ABB RAPID module: Arm_Weld

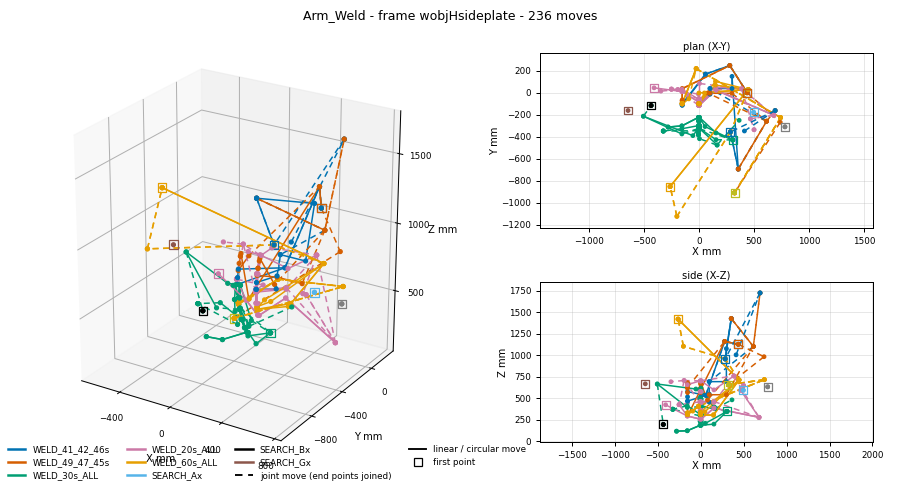
[picture p0: tool path of Arm_Weld in frame wobjHsideplate, 236 of 1587 moves have a stored position in this frame; points joined in program order, loops and branches not executed]
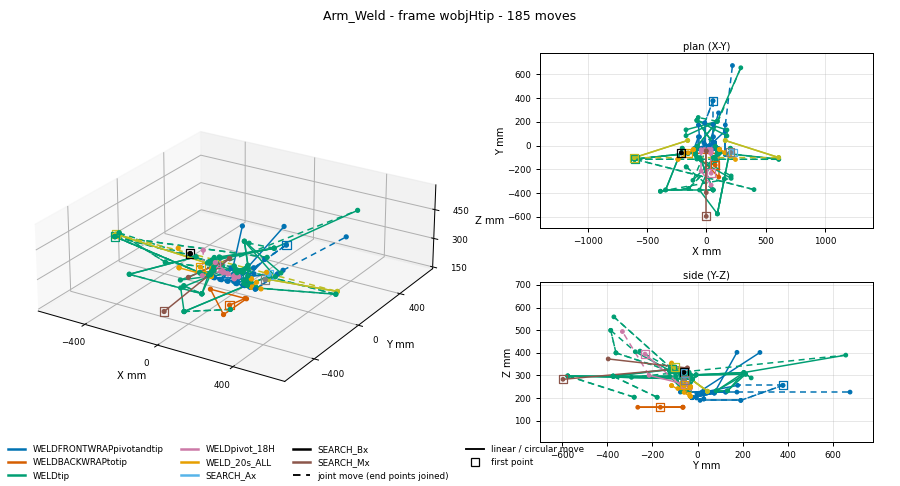
[picture p1: tool path of Arm_Weld in frame wobjHtip, 185 of 1587 moves have a stored position in this frame; points joined in program order, loops and branches not executed]
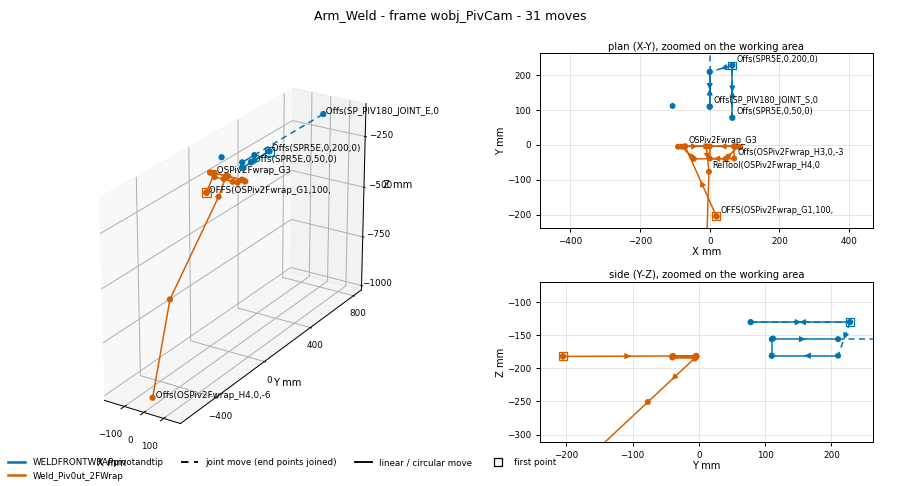
[picture p2: tool path of Arm_Weld in frame wobj_PivCam, 31 of 1587 moves have a stored position in this frame; points joined in program order, loops and branches not executed]
MODULE W6806128_R4_PR3

!!!!!! this is the 7th revision of integrating the NEW PivCAM stuff  SY 12-06-18!!!
!!!!!!THIS IS A PR3 TEMPLATE PROGRAM FOR 18H SIP lesspoints (928)!!!!!03-02-20!!!SY!!!
!!!!!! HAS 3 points 60s!!!
!!!!!!  CAME FROM EMPTY ARM 03-02-20!!!!!!!!
!!!!!! LAYED OUT TO WORK WITH Assembly_Data R12.sys 04-08-18!!!!!!
!!!!!!HAS R100!!04-08-18!!!!!!
!!!!!!!!!BORN FROM 6935130 18H!!!!!!!!
!!!!!!HAS SEARCH_Mx, SEARCH_Lx, SEARCH_Ax, SEARCH_Bx, SEARCH_Gx, SEARCH_Hx!!!!!!!!!!
!!!!!!HAS ZERO_X_A_ALL,ZERO_X_B_ALL,ZERO_X_G_ALL,ZERO_X_H_ALL,ZERO_X_L_ALL,ZERO_X_M_ALL,!!!!!!!!!!
!!!!!!THIS TEMPLATE HAS BEEN REVIEWED IN 5.61  03-02-20!!!!!!!
!!!!!!!!!18H!!!!!!!!!!!!!
!!!!!!!!has FBadjpos/UNtilt19!!! 04-08-18!!!!!
!!!!!!!! HAS TBR/L!04-08-18!!!!!!!!!!!
!!!!!!...04-08-18.now HAS nozzle searching w/IF!!!!!!!
!!!!!!!..anchor is SIP nozzle searching FOR H_ANCHOR,TAPERED_SQUARE_ANCHOR, PLAIN SQUARE ANCHOR....01-09-18!!!!!!!!!!
!!!!!!!Nozzle searching on Anchor is pointing TIP.....(short Wotox)(1012)....08-28-18!!!!!!!!!!
!!!!!!! Fixed a wart in the weld_all_PJ proc....wrong callout in a seamparam in a joint search....03-25-18!!!!
!!!!!!! Created a new x plotter for the anchor (SET_ANCHOR_X) with input 04-08-18
!!!!!!! Created a new x pose SR_AHF_X,SR_AHG_X for the anchor procs  04-08-18
!!!!!!! Created new robtargets  SP_AGFX_E SP_AGFX_S SP_AHFX_E SP_AGFX_S for the anchor procs  04-08-18
!!!!!!! REVISED ALL ANCHOR PROCS TO ADD X SEARCHES ON FRONT and BACK 04-08-18
!!!!!!! ADDED THE PIV PROCs that got Revised 04-08-18
!!!!!!! CUT AND PASTE WELDATA INTO here from template 12-06-18!!!!!!!
!!!!!!! has WELDpivot_18H (only two passes!) 08-16-18!!!!
!!!!!!! now with TWO PASSES ON THE TIP!!!!!!!!!!!!!!!
!!!!!!!HAS dripstop_A and_G with IF...11-27-19!!!!!!!!
!!!!!!! added z_RESETS 04-22-19!!!!!!!!!!!!!!!!!!!!!
!!!!!!!! added ADJWrapperROOTWIDTH18H 11-18-19!!!!!!!!!!!
!!!!!!!!Killed the 0.5 WaitTime in dots in Weldpivot 01-16-20!!!!!!!!
!!!!!!!!!03-02-20 Uses the Revised (R2) Pivot plotter for 18H!!!!!!
!!!!!!!!! 09-28-20 TRACKING HEIGHT ONLY ON ABTBL,ABTBR,GHTBL,GHTBR!!!!!!!!!!




    PERS num scoot_G:=-2.3;
    PERS num scoot_A:=3;

   PERS pose SRRY1:=[[-0.278763,0,0],[1,0,0,0]];

    PERS num THISPROGRAM:=6806128;
    PERS num THISPARTREV:=4;
    PERS num THISPROGREV:=3;
    PERS num THISPROGPREP:=191118;
    VAR bool bSIP:=TRUE;
    VAR bool bINTEGRAL_TIP:=FALSE;
    VAR bool bANC2CLOSE2_TIP:=FALSE;
    VAR bool bBACK_STEP:=FALSE;
    VAR bool bFEEDBACK:=FALSE;
    PERS num THISproglastchanged:=200928;
    VAR bool bUnderANCHOR:=TRUE;
    VAR bool bmissweld:=FALSE;
    VAR num reg100:=0;

!!!!!!!!!!!!!!!!!!!!!!!!!!!!!!!!!  vvvv THESE WELD AND TRACKDATAS COPIED INTO TEMPLATE 11-29-18 vvv !!!!!!!!!!!!!!!!!!!!!!!!!!!!!!!!!!!!
 !!!!!!!!!!!!!!!!WE WILL CALL THIS 18H (8mm) wrapper data!!!!!!!
!!!!!!!!!!dropped current targets to proper values 11-29-18!!!!!!!!!
!!!!!!!!11-29-18!!!!!!!!!!!!


    TASK PERS seamdata smpqroot:=[1,2,[5,5,27.5,135.467,0,325,0,0,0],0,0,0,0,0,[0,0,0,0,0,0,0,0,0],2,0.5,[5,5,27.5,139.7,0,325,0,0,0],0.08,0,[0,0,0,0,0,0,0,0,0],3];
    TASK PERS welddata wdP1Q1root:=[9.31333,0,[5,5,27.5,156.633,0,325,0,0,0],[0,0,0,0,0,0,0,0,0]];

    TASK PERS trackdata trABTBR3:=[0,FALSE,25,[5,40,40,0,-3,0,0,0,0],[0,0,0,0,0,0,0]];
    TASK PERS trackdata trGHTBR3:=[0,FALSE,25,[5,40,40,0,-3,0,0,0,0],[0,0,0,0,0,0,0]];


    PERS num percentcoverpass:=39;
    PERS num percentrootpass:=35;
    PERS num percent2pass:=40;

	TASK PERS trackdata trLM10hiteonly:=[0,FALSE,25,[5,40,40,0,0,0,0,0,0],[0,0,0,0,0,0,0]];

    TASK PERS trackdata trPJhiteonly1:=[0,TRUE,25,[5,40,40,0,0,0,0,0,0],[0,0,0,0,0,0,0]];
    TASK PERS welddata wdGH_CAM_PJ_ROOTfast:=[5.08,0,[5,0,27.8,139.7,0,325,0,0,0],[0,0,0,0,0,0,0,0,0]];
    TASK PERS welddata wdGH_RND_PJ_ROOTfast:=[5.08,0,[5,0,27.8,143.933,0,325,0,0,0],[0,0,0,0,0,0,0,0,0]];
    TASK PERS welddata wdGH_RND_PJ_ROOT:=[3.38667,0,[5,0,27.8,139.7,0,325,0,0,0],[0,0,0,0,0,0,0,0,0]];
    TASK PERS welddata wdGH_CAM_PJ_ROOT:=[3.38667,0,[5,0,27.8,148.167,0,325,0,0,0],[0,0,0,0,0,0,0,0,0]];
    TASK PERS welddata wdGH_RND_PJ_CVR:=[2.96333,0,[5,5,27.5,143.933,0,325,0,0,0],[0,0,0,0,0,0,0,0,0]];

     TASK PERS welddata wdGH_CAM_PJ_FILL1:=[3.38667,0,[5,5,27.8,148.167,0,325,0,0,0],[0,0,0,0,0,0,0,0,0]];
     TASK PERS welddata wdGH_CAM_PJ_FILL2:=[3.38667,0,[5,5,27.8,148.167,0,325,0,0,0],[0,0,0,0,0,0,0,0,0]];
     TASK PERS welddata wdGH_CAM_PJ_CVR:=[3.38667,0,[5,5,27.8,148.167,0,325,0,0,0],[0,0,0,0,0,0,0,0,0]];

     TASK PERS weavedata wvGH_CAM_PJ_FILL2:=[1,0,3,3,0,0.2,0,0.2,0,0,0,0,0,0,0];
     TASK PERS weavedata wvGH_CAM_PJ_FILL1:=[1,0,3,3,0,0.2,0,0.2,0,0,0,0,0,0,0];
     TASK PERS weavedata wvGH_CAM_PJ_CVR:=[1,0,3,3,0,0.2,0,0.2,0,0,0,0,0,0,0];
	 TASK PERS weavedata wvGH_RND_PJ_CVR:=[1,0,5,5,0,0.2,0,0.2,0,0,0,0,0,0,0];

    TASK PERS seamdata smGH_RND_PJ:=[1,2,[5,5,27.8,148.167,0,325,0,0,0],0,1,0,0,0,[0,0,0,0,0,0,0,0,0],1.5,1.3,[5,5,27.8,148.167,0,325,0,0,0],0.08,0,[0,0,0,0,0,0,0,0,0],1];
    TASK PERS seamdata smGH_CAM_PJ:=[1,2,[5,5,27.8,148.167,0,325,0,0,0],0,1,0,0,0,[0,0,0,0,0,0,0,0,0],1.5,1.3,[5,5,27.8,148.167,0,325,0,0,0],0.08,0,[0,0,0,0,0,0,0,0,0],1];

	TASK PERS trackdata trGH:=[0,FALSE,25,[0,40,40,0,0,0,0,0,0],[0,0,0,0,0,0,0]];
	TASK PERS trackdata trAB:=[0,FALSE,25,[0,40,40,0,0,0,0,0,0],[0,0,0,0,0,0,0]];

    TASK PERS trackdata trABTBR:=[0,FALSE,25,[5,40,40,0,-1,0,0,0,0],[0,0,0,0,0,0,0]];
    TASK PERS trackdata trABTBL:=[0,FALSE,25,[5,40,40,0,1,0,0,0,0],[0,0,0,0,0,0,0]];
    TASK PERS trackdata trGHTBR:=[0,FALSE,25,[5,40,40,0,-1,0,0,0,0],[0,0,0,0,0,0,0]];
    TASK PERS trackdata trGHTBL:=[0,FALSE,25,[5,40,40,0,1,0,0,0,0],[0,0,0,0,0,0,0]];


    TASK PERS trackdata trLM18cast:=[0,FALSE,25,[0,40,30,0,0,0,0,0,0],[0,0,0,0,0,0,0]];
    TASK PERS trackdata trTIPears:=[0,FALSE,25,[5,40,40,0,0,0,0,0,0],[0,0,0,0,0,0,0]];
	TASK PERS trackdata trRS56:=[0,TRUE,50,[5,40,40,0,0,0,0,0,0],[0,0,0,0,0,0,0]];
	TASK PERS trackdata trHCYLANCHhiteonly:=[0,TRUE,25,[0,40,40,0,0,0,0,0,0],[0,0,0,0,0,0,0]];
	TASK PERS trackdata track0:=[0,FALSE,0,[0,0,0,0,0,0,0,0,0],[0,0,0,0,0,0,0]];
	TASK PERS trackdata trLM10:=[0,FALSE,25,[0,50,30,0,0,0,0,0,0],[0,0,0,0,0,0,0]];
	TASK PERS trackdata trTIPBACKhiteonly:=[0,TRUE,25,[5,40,40,0,0,0,0,0,0],[0,0,0,0,0,0,0]];

    TASK PERS welddata wdGH195tip:=[6.64633,0,[5,5,26.8,127,0,305,0,0,0],[0,0,0,0,0,0,0,0,0]];
    TASK PERS weavedata wvGH195tip:=[1,0,2,2,0,0,0,0,0,0,0,0,0,0,0];

    TASK PERS welddata wdGH29tip:=[6.68867,0,[5,5,26.8,127,0,305,0,0,0],[0,0,0,0,0,0,0,0,0]];
    TASK PERS weavedata wvGH29tip:=[1,0,2,2,0,0,0,0,0,0,0,0,0,0,0];

	TASK PERS seamdata smGH195:=[1,2,[5,5,27.5,122.767,0,290,0,0,0],0,1,0,0,0,[0,0,0,0,0,0,0,0,0],2,0.8,[5,5,27,122.767,0,290,0,0,0],0.08,0,[0,0,0,0,0,0,0,0,0],2];
	TASK PERS welddata wdGH195:=[6.68867,0,[5,5,26.8,127,0,305,0,0,0],[0,0,0,0,0,0,0,0,0]];
	TASK PERS weavedata wvGH195:=[1,0,2,2,0,0,0,0,0,0,0,0,0,0,0];
	TASK PERS weavedata wvGH29:=[1,0,2,2,0,0,0,0,0,0,0,0,0,0,0];
	TASK PERS seamdata smGH29:=[1,2,[5,5,27.3,122.767,0,290,0,0,0],0,1,0,0,0,[0,0,0,0,0,0,0,0,0],1.3,0.9,[5,5,27,122.767,0,290,0,0,0],0.08,0,[0,0,0,0,0,0,0,0,0],2];
	TASK PERS welddata wdGH29:=[6.68867,0,[5,5,26.8,127,0,305,0,0,0],[0,0,0,0,0,0,0,0,0]];

	TASK PERS welddata wdGH40A:=[5.92667,0,[5,5,27.5,139.7,0,325,0,0,0],[0,0,0,0,0,0,0,0,0]];
	TASK PERS seamdata smGH40A:=[1,2,[5,5,27.5,139.7,0,325,0,0,0],0,1,0,0,0,[0,0,0,0,0,0,0,0,0],3,1,[5,5,27.5,139.7,0,325,0,0,0],0.08,0,[0,0,0,0,0,0,0,0,0],2];
	TASK PERS weavedata wvGH40A:=[1,0,2,2,0,0,0,0,0,0,0,0,0,0,0];

	TASK PERS weavedata wvGH40B:=[1,0,2,2,0,0,0,0,0,0,0,0,0,0,0];
	TASK PERS welddata wdGH40B:=[4.65667,0,[5,5,27.5,139.7,0,325,0,0,0],[0,0,0,0,0,0,0,0,0]];

	TASK PERS welddata wdGH40C:=[7.62,0,[5,5,27.5,143.933,0,325,0,0,0],[0,0,0,0,0,0,0,0,0]];

	TASK PERS welddata wdGH40F:=[7.62,0,[5,0,27.5,131.233,0,300,0,0,0],[0,0,0,0,0,0,0,0,0]];
	TASK PERS seamdata smGH40F:=[1,1,[5,0,27.5,127,0,300,0,0,0],0,1,0,0,0,[0,0,0,0,0,0,0,0,0],1,0,[0,0,0,0,0,0,0,0,0],0,0,[0,0,0,0,0,0,0,0,0],0];

!!!!!!!!!!!!!!!!!BEST 18H weldata and beveldata as of 11-29-18 !!!!!!

	TASK PERS welddata wdR1R2root:=[11.0067,0,[5,5,27.5,152.4,0,320,0,0,0],[0,0,0,0,0,0,0,0,0]];
    TASK PERS weavedata wvRSroot:=[1,0,6,1,0,0,0,0,0,0,0,0,0,0,0];
	TASK PERS welddata wdR5R6cover:=[3.38667,0,[5,5,27.5,143.933,0,325,0,0,0],[0,0,0,0,0,0,0,0,0]];
	TASK PERS welddata wdP1Q1cover:=[4.65667,0,[5,5,27.5,143.933,0,325,0,0,0],[0,0,0,0,0,0,0,0,0]];
	TASK PERS weavedata wvR5R6cover:=[1,0,2,3,0,0.1,0,0.1,0,0,0,0,0,0,0];
	TASK PERS weavedata wvP1Q1cover:=[1,0,2,2,0,0.1,0,0.1,0,20,0,0,0,0,0];
	TASK PERS seamdata smPQRS:=[1,2,[5,5,27.5,148.167,0,320,0,0,0],0,1,0,0,0,[0,0,0,0,0,0,0,0,0],1.2,1.2,[5,5,27.5,139.7,0,320,0,0,0],0.08,0,[0,0,0,0,0,0,0,0,0],1];
	TASK PERS seamdata smPQRSroot:=[1,2,[5,5,27.8,148.167,0,325,0,0,0],0,1,0,0,0,[0,0,0,0,0,0,0,0,0],0,0,[5,5,27.5,127,0,325,0,0,0],0.08,0,[0,0,0,0,0,0,0,0,0],1];
	TASK PERS seamdata smRS1:=[1,2,[5,5,27.5,148.167,0,320,0,0,0],0,1,0,0,0,[0,0,0,0,0,0,0,0,0],1.2,1.2,[5,5,27.5,139.7,0,320,0,0,0],0.08,0,[0,0,0,0,0,0,0,0,0],1];
	TASK PERS seamdata smPQ1:=[1,2,[5,5,27.5,148.167,0,320,0,0,0],0,1,0,0,0,[0,0,0,0,0,0,0,0,0],1.2,1.2,[5,5,27.5,139.7,0,320,0,0,0],0.08,0,[0,0,0,0,0,0,0,0,0],1];

	TASK PERS welddata wdGH1thru8:=[5.50333,0,[5,5,27.5,139.7,0,315,0,0,0],[0,0,0,0,0,0,0,0,0]];
	TASK PERS seamdata smGH1thru8:=[1,2,[5,5,27.5,143.933,0,320,0,0,0],0,1,0,0,0,[0,0,0,0,0,0,0,0,0],1,1.6,[5,5,27.5,143.933,0,320,0,0,0],0.08,0,[0,0,0,0,0,0,0,0,0],1.5];
	TASK PERS weavedata wvGH1thru8:=[1,0,2,2,0,0,0,0,0,0,0,0,0,0,0];

	TASK PERS seamdata smLM10:=[1,2,[5,5,27.5,139.7,0,320,0,0,0],0,1,0,0,0,[0,0,0,0,0,0,0,0,0],1.3,1.2,[5,5,27.5,127,0,320,0,0,0],0.08,0,[0,0,0,0,0,0,0,0,0],1];
	TASK PERS welddata wdLM10:=[5.50333,0,[5,5,27.5,135.467,0,310,0,0,0],[0,0,0,0,0,0,0,0,0]];
	TASK PERS weavedata wvLM10:=[1,0,2,2,0,0,0,0,0,0,0,0,0,0,0];

	TASK PERS seamdata smTU:=[1,2,[5,5,27.5,135.467,0,320,0,0,0],0,1,0,0,0,[0,0,0,0,0,0,0,0,0],1.5,1.5,[5,5,27.5,139.7,0,320,0,0,0],0.08,0,[0,0,0,0,0,0,0,0,0],1.5];
	TASK PERS welddata wdT1112cover:=[4.445,0,[5,5,27.5,143.933,0,325,0,0,0],[0,0,0,0,0,0,0,0,0]];
	TASK PERS weavedata wvT1112cover:=[1,0,2,4,0,0.1,0,0.1,0,0,0,0,0,0,0];

	TASK PERS seamdata smTU2122:=[1,2,[5,5,27.3,148.167,0,325,0,0,0],0,1,0,0,0,[0,0,0,0,0,0,0,0,0],1.5,1,[5,5,27.3,127,0,325,0,0,0],0.08,0,[0,0,0,0,0,0,0,0,0],1];
	TASK PERS welddata wdTU2122cover:=[3.81,0,[5,5,27.75,141.817,0,325,0,0,0],[0,0,0,0,0,0,0,0,0]];
	TASK PERS weavedata wvTU2122cover:=[1,0,2,4,0,0.2,0,0.2,0,0,0,0,0,0,0];


    TASK PERS welddata wdTU3031root:=[6.77333,0,[5,5,27.5,135.467,0,325,0,0,0],[0,0,0,0,0,0,0,0,0]];
	TASK PERS seamdata smTU3031:=[1,2,[5,5,27.5,139.7,0,325,0,0,0],0,1,0,0,0,[0,0,0,0,0,0,0,0,0],3,1.2,[5,5,27.5,139.7,0,325,0,0,0],0.08,0,[0,0,0,0,0,0,0,0,0],2];
	TASK PERS welddata wdTU3031cover:=[2.96333,0,[5,5,27.5,143.933,0,325,0,0,0],[0,0,0,0,0,0,0,0,0]];
	TASK PERS weavedata wvTU3031cover:=[1,0,2,4,0,0.1,0,0.1,0,0,0,0,0,0,0];

    TASK PERS seamdata smTU3031quick:=[1,2,[5,5,27.5,135.467,0,325,0,0,0],0,1,0,0,0,[0,0,0,0,0,0,0,0,0],3,1,[5,5,27.5,135.467,0,325,0,0,0],0.08,0,[0,0,0,0,0,0,0,0,0],1.6];
    TASK PERS welddata wdTU3031quick:=[4.65667,0,[5,5,27.5,143.933,0,325,0,0,0],[0,0,0,0,0,0,0,0,0]];
    TASK PERS weavedata wvTU3031quick:=[1,0,2,2,0,0.2,0,0.2,0,0,0,0,0,0,0];

    TASK PERS seamdata smTU3031quick2:=[1,2,[5,5,27.5,139.7,0,325,0,0,0],0,1,0,0,0,[0,0,0,0,0,0,0,0,0],3,1.2,[5,5,27.5,139.7,0,325,0,0,0],0.08,0,[0,0,0,0,0,0,0,0,0],2];
    TASK PERS welddata wdTU3031quick2:=[3.937,0,[5,5,27.5,143.933,0,325,0,0,0],[0,0,0,0,0,0,0,0,0]];
    TASK PERS weavedata wvTU3031quick2:=[1,0,2,2,0,0,0,0,0,0,0,0,0,0,0];

    TASK PERS welddata wdTU3031quick3:=[3.175,0,[5,5,27.5,143.933,0,325,0,0,0],[0,0,0,0,0,0,0,0,0]];

     TASK PERS welddata wdTU3031SLOW:=[3.38667,0,[5,5,27.5,143.933,0,325,0,0,0],[0,0,0,0,0,0,0,0,0]];
    TASK PERS weavedata wvTU3031SLOW:=[1,0,2,4,0,0,0,0,0,0,0,0,0,0,0];
    TASK PERS seamdata smTU3031SLOW:=[1,2,[5,5,27.5,139.7,0,330,0,0,0],0,1,0,0,0,[0,0,0,0,0,0,0,0,0],3,1.2,[5,5,27.5,139.7,0,325,0,0,0],0.08,0,[0,0,0,0,0,0,0,0,0],2];

	TASK PERS seamdata smT50:=[1,1,[5,0,27,135.467,0,320,0,0,0],0,1,0,0,0,[0,0,0,0,0,0,0,0,0],2,1.2,[5,5,27,139.7,0,325,0,0,0],0,0,[0,0,0,0,0,0,0,0,0],2];
	TASK PERS welddata wdT50:=[4.23333,0,[5,0,27,139.7,0,325,0,0,0],[0,0,0,0,0,0,0,0,0]];
	TASK PERS weavedata wvT50:=[1,0,2,6,0,0,0,0,0,0,0,0,0,0,0];
    TASK PERS welddata wdT50root:=[6.35,0,[5,0,27.5,169.333,0,325,0,0,0],[0,0,0,0,0,0,0,0,0]];

    TASK PERS seamdata smTU7071:=[1,2,[5,5,27.5,148.167,0,320,0,0,0],0,0,0,0,0,[0,0,0,0,0,0,0,0,0],1.5,1.5,[5,5,27.5,143.933,0,325,0,0,0],0.08,0,[0,0,0,0,0,0,0,0,0],1];
    TASK PERS welddata wdTU7071:=[2.96333,0,[5,5,27.5,143.933,0,325,0,0,0],[0,0,0,0,0,0,0,0,0]];
    TASK PERS weavedata wvTU7071:=[1,0,2,3.5,0,0.3,0,0.3,0,0,0,0,0,0,0];

    TASK PERS seamdata smTUroot:=[1,2,[5,5,27,148.167,0,325,0,0,0],0,1,0,0,0,[0,0,0,0,0,0,0,0,0],1.5,0,[5,5,27,139.7,0,325,0,0,0],0.08,0,[0,0,0,0,0,0,0,0,0],1.5];
    TASK PERS welddata wdT1112root:=[8.46667,0,[5,5,27.5,169.333,0,325,0,0,0],[0,0,0,0,0,0,0,0,0]];

	TASK PERS seamdata smHCYLANCH:=[1,2,[5,5,27.5,131.233,0,325,0,0,0],0,1,0,0,0,[0,0,0,0,0,0,0,0,0],1.5,1,[5,5,27.5,127,0,325,0,0,0],0.08,0,[0,0,0,0,0,0,0,0,0],1];
	TASK PERS welddata wdHCYLANCH:=[3.81,0,[5,5,27.5,143.933,0,325,0,0,0],[0,0,0,0,0,0,0,0,0]];
	TASK PERS weavedata wvHCYLANCH:=[1,0,2,2,0,0.1,0,0.1,0,0,0,0,0,0,0];

    PERS edgedata edgedata_HRND_PJ:=[0,8,3,0.052];
    PERS edgedata edgedata_GRND_PJ:=[0,8,3,0.052];
    PERS edgedata edgedata_GCAM_PJ:=[0,8,3,0.052];
    PERS edgedata edgedata_HCAM_PJ:=[0,8,3,0.052];

    TASK PERS seamparam seampar_HRND_PJ:=["H_PJ",0,[42,0.052,339.999,0,0,1,11,0,4,14,-6,2,15,250],202.66,14.4757,14.4757];
    TASK PERS seamparam seampar_GRND_PJ:=["G_PJ",0,[45,0.052,339.999,0,0,1,11,0,4,14,-6,2,15,250],198.028,14.1448,14.1448];
    TASK PERS seamparam seampar_GCAM_PJ:=["G_PJ",0,[40,0.052,148.167,0,0,1,11,0,3,11,-7,2,100,500],179.688,14.7105,10.9592];
    TASK PERS seamparam seampar_HCAM_PJ:=["H_PJ",0,[40,0.052,350.001,0,0,1,11,0,3,11,-7,2,100,500],184.46,15.0514,11.3001];

    PERS bevelparam bevelparam_HRND_pJ:=[6,0,20,0,14,14,0,5,0,0,15,2,2,0.052];
    PERS bevelparam bevelparam_HCAM_pJ:=[4,0,15,0,14,14,0,5,0,0,15,2,2,0.052];
    PERS bevelparam bevelparam_GRND_pj:=[6,0,20,0,14,14,0,5,0,0,15,2,2,0.052];
    PERS bevelparam bevelparam_GCAM_pj:=[4,0,15,0,14,14,0,5,0,0,15,2,2,0.052];

!!!@######################################################################
!  weld datas for the piv "B" weld  18H
    TASK PERS seamdata smJK:=[1,2,[5,5,27.5,139.7,0,325,0,0,0],0,1,0,0,0,[0,0,0,0,0,0,0,0,0],0.5,0.5,[5,5,27.5,127,0,325,0,0,0],0.08,0,[0,0,0,0,0,0,0,0,0],1.2];
    TASK PERS welddata wdJK:=[4.23333,0,[5,5,27.5,143.933,0,325,0,0,0],[0,0,0,0,0,0,0,0,0]];
    TASK PERS weavedata wvJK:=[1,0,2,4,0,0,0,0,0,0,0,0,0,0,0];
    TASK PERS seamdata smJKnofill:=[1,2,[5,5,27.5,139.7,0,325,0,0,0],0,1,0,0,0,[0,0,0,0,0,0,0,0,0],2,0.8,[5,5,27.5,127,0,300,0,0,0],0.08,0,[0,0,0,0,0,0,0,0,0],2];
    TASK PERS welddata wdJK1:=[5.92667,0,[5,5,27.5,135.467,0,330,0,0,0],[0,0,0,0,0,0,0,0,0]];
    TASK PERS seamdata smJK1:=[1,2,[5,5,27.5,139.7,0,330,0,0,0],0,1,0,0,0,[0,0,0,0,0,0,0,0,0],0.5,0.5,[5,5,27.5,127,0,325,0,0,0],0.08,0,[0,0,0,0,0,0,0,0,0],1.2];
    TASK PERS welddata wdJKroot:=[6.77333,0,[5,0,27,131.233,0,310,0,0,0],[0,0,0,0,0,0,0,0,0]];
    TASK PERS seamdata smJKroot:=[2,2,[5,0,27,135.467,0,320,0,0,0],0,1,0,0,0,[0,0,0,0,0,0,0,0,0],2,0,[5,0,0,0,0,0,0,0,0],0,0,[0,0,0,0,0,0,0,0,0],2];
    TASK PERS weavedata wvJKroot:=[1,0,2,1,0,0,0,0,0,0,0,0,0,0,0];


    !!!!!!!!!!!!!!!!!!!!!!!!!!!!!!!!!!Nums for groove searches!!!!!!!!!!!!!!!!!!!!!!!!!!!!!!!!!
VAR num width_T11:=0;
VAR num width_G50:=0;
VAR num width_H50:=0;
VAR num width_RSR1:=0;
VAR num width_PQ1:=0;
VAR num width_T50:=0;
VAR num width_T40:=0;

PERS num Rrootarea:=0;
PERS num GH50rootarea:=0;
VAR num reg7:=0;
VAR num reg8:=0;

PERS edgeresult edgeresultT11:=[[[0.0793076,-0.129463,0.364746],[1,0,0,0]],[[0.0793076,-0.129461,0.364738],[1,0,0,0]],[93.0493,-36.0195,105.505],[93.1546,-28.1059,106.673]];
PERS edgeresult edgeresultT50:=[[[0.0793076,-0.129463,0.364746],[1,0,0,0]],[[0.0793076,-0.129461,0.364738],[1,0,0,0]],[93.0493,-36.0195,105.505],[93.1546,-28.1059,106.673]];
PERS edgeresult edgeresultT40:=[[[0.0793076,-0.129463,0.364746],[1,0,0,0]],[[0.0793076,-0.129461,0.364738],[1,0,0,0]],[93.0493,-36.0195,105.505],[93.1546,-28.1059,106.673]];

PERS bevelparam bevelparamT50:=[8,0,0,0,5,5,0,0,10,0,10,0,0,0.052];
PERS bevelparam bevelparamR1:=[5,0,30,180,8,8,0,0,0,0,5,0,3,0.052];
PERS bevelparam bevelparamA100:=[5,2,2,180,12.7,12.7,0,0,0,0,12.7,0,4,0.052];

PERS edgedata edgedataT55:=[0,8,3,0.052];
PERS edgedata edgedataR10:=[1,8,3,0.052];
PERS edgedata edgedataPQ1:=[0,8,3,0.052];
PERS edgedata edgedataT50:=[0,8,3,0.052];
PERS edgedata edgedataT40:=[0,8,3,0.052];

TASK PERS seamparam seamparT50:=["TWELD",0,[70,0.052,340,0,0,1,11,0,3.5,8,0,2,15,100],82.8542,10.8629,0.862882];
TASK PERS seamparam seamparR1:=["RWELD",0,[80,0.052,340,0,0,1,11,0,2,13,-2,2,25,135],24.4145,5.36121,0.74241];
TASK PERS seamparam seamparS1:=["SWELD",0,[80,0.052,340,0,0,1,11,0,2,13,-2,2,25,135],24.4145,5.36121,0.74241];

TASK PERS layerdata layRWELD:=["RWELD",[78,0.052,340,0,0,1,11,0,0.5,14,0,2,40,125],[1,0,0,0,0,10,0,0,0,0,0,0,[0,0,0,0,0,0]]];
TASK PERS layerdata laySWELD:=["SWELD",[78,0.052,340,0,0,1,11,0,0.5,11,0,2,40,125],[1,0,0,0,0,10,10,0,0,0,0,0,[0,0,0,0,0,0]]];
!!!!!!!!!!!!!!!!!!!!!!!!!!!!!!!!!  ^^^^THESE DATAS COPIED INTO TEMPLATE 11-29-18 PTL ^^^^^^!!!!!!!!!!!!!!!!!!!!!!!!!!!!!!!!!!!!
!!!!!!!!!!!!!!!!!!!!!!!!!!!!!!!!!  ^^^^THESE WELD AND TRACKDATAS COPIED INTO TEMPLATE 11-29-18  ^^^^^^!!!!!!!!!!!!!!!!!!!!!!!!!!!!!!!!!!!!

    !  this rob target is for setting the YZ components of X-Searches
    PERS robtarget PIV_YZ_MASTER_SEARCH:=[[0.08,-16.55,-269.25],[0.410879,-0.609379,0.562263,0.379072],[-1,0,0,0],[9E+09,-0.000202659,0.00203972,9E+09,9E+09,9E+09]];

  !PIVOT_CAM_LOBE
    PERS robtarget H_RND_1:=[[138.75,-56.15,-128.81],[0.791215,-0.426463,-0.392456,0.195157],[-1,1,-2,0],[9E+09,8.53587,-48.4641,9E+09,9E+09,9E+09]];
	PERS robtarget H_RND_2:=[[138.75,-52.19,-134.16],[0.790823,-0.424031,-0.394665,0.197577],[-1,1,-2,0],[9E+09,8.53587,-48.4642,9E+09,9E+09,9E+09]];
	PERS robtarget H_RND_3:=[[138.75,-6.71,-203.72],[0.77354,-0.424849,-0.422397,0.206687],[-1,1,-2,0],[9E+09,8.53592,-48.464,9E+09,9E+09,9E+09]];
	PERS robtarget H_RND_4:=[[138.76,-1.73,-209.20],[0.831387,-0.307692,-0.395259,0.240606],[-1,1,-3,0],[9E+09,8.5359,-60,9E+09,9E+09,9E+09]];
	PERS robtarget H_RND_5:=[[138.77,4.77,-209.99],[0.825767,-0.235199,-0.422961,0.289645],[-1,1,-3,0],[9E+09,17.3096,-65,9E+09,9E+09,9E+09]];
	PERS robtarget H_RND_6:=[[138.76,19.31,-210.84],[0.84569,-0.248028,-0.384006,0.275373],[-1,1,-3,0],[9E+09,17.3096,-67,9E+09,9E+09,9E+09]];
	PERS robtarget H_RND_7:=[[138.75,20.19,-212.40],[0.714518,-0.516691,-0.337745,0.329276],[0,2,-3,0],[9E+09,-11.563,-48.937,9E+09,9E+09,9E+09]];
	PERS robtarget H_RND_8:=[[138.01,1.53,-260.75],[0.775065,-0.4237,-0.381985,0.271739],[-1,2,-3,0],[9E+09,-18.82,-50,9E+09,9E+09,9E+09]];

    PERS robtarget G_RND_1:=[[-137.19,-60.62,-128.24],[0.743875,-0.503842,0.273771,-0.34328],[-1,1,-2,0],[9E+09,8.53587,48.4641,9E+09,9E+09,9E+09]];
	PERS robtarget G_RND_2:=[[-137.17,-55.07,-134.19],[0.733198,-0.515384,0.284408,-0.340458],[-1,1,-2,0],[9E+09,8.53596,48.4639,9E+09,9E+09,9E+09]];
	PERS robtarget G_RND_3:=[[-137.16,-8.79,-203.74],[0.739724,-0.505179,0.29895,-0.328986],[-1,1,-2,0],[9E+09,8.53588,48.4641,9E+09,9E+09,9E+09]];
	PERS robtarget G_RND_4:=[[-137.17,-4.28,-209.04],[0.79307,-0.400763,0.274228,-0.367733],[-1,1,-3,0],[9E+09,8.5359,60,9E+09,9E+09,9E+09]];
	PERS robtarget G_RND_5:=[[-137.17,4.80,-210.46],[0.793114,-0.347997,0.30544,-0.395695],[-1,1,-3,0],[9E+09,17.3096,65,9E+09,9E+09,9E+09]];
	PERS robtarget G_RND_6:=[[-137.17,17.37,-210.42],[0.775238,-0.392589,0.31475,-0.381854],[-1,1,-2,0],[9E+09,17.3096,66.9999,9E+09,9E+09,9E+09]];
	PERS robtarget G_RND_7:=[[-137.15,18.66,-210.61],[0.703635,-0.503523,0.333985,-0.37392],[-1,1,-3,0],[9E+09,-11.563,48.937,9E+09,9E+09,9E+09]];
	PERS robtarget G_RND_8:=[[-137.9,0.7,-261.77],[0.695401,-0.476371,0.308489,-0.440823],[-1,1,-3,0],[9E+09,18.82,50.0001,9E+09,9E+09,9E+09]];

	PERS robtarget G_CAM_1:=[[-92.072,-56.19,-102.39],[0.7891,-0.350678,-0.49169,-0.112189],[-1,1,-2,0],[9E+09,-4.99999,-46.4189,9E+09,9E+09,9E+09]];
	PERS robtarget G_CAM_2:=[[-92.072,-45.7,-130.82],[0.78473,-0.351653,-0.498636,-0.109091],[-1,1,-2,0],[9E+09,-4.99999,-46.4189,9E+09,9E+09,9E+09]];
	PERS robtarget G_CAM_3:=[[-92.072,-38.95,-140.06],[0.856961,-0.220645,-0.451261,-0.115311],[-1,0,-2,0],[9E+09,12,-58,9E+09,9E+09,9E+09]];
	PERS robtarget G_CAM_4:=[[-92.072,-16.92,-148.25],[0.84678,-0.238772,-0.459157,-0.122986],[-1,0,-2,0],[9E+09,14,-60,9E+09,9E+09,9E+09]];
	PERS robtarget G_CAM_5:=[[-92.072,-12.59,-151.76],[0.776964,-0.265744,-0.537769,-0.191078],[-1,0,-2,0],[9E+09,-2.00001,-50.0003,9E+09,9E+09,9E+09]];
	PERS robtarget G_CAM_6:=[[-92.072,-13.07,-165.64],[0.665852,-0.294079,-0.652518,-0.210665],[-1,0,-2,0],[9E+09,-15,-54.9999,9E+09,9E+09,9E+09]];
	PERS robtarget G_CAM_7:=[[-92.072,-12.78,-181.52],[0.705791,-0.252132,-0.619909,-0.232383],[-1,0,-2,0],[9E+09,-18,-54.9998,9E+09,9E+09,9E+09]];
	PERS robtarget G_CAM_8:=[[-92.072,-1.59,-188.14],[0.802926,-0.25985,-0.496077,-0.204193],[-1,0,-2,0],[9E+09,3.00002,-55.0003,9E+09,9E+09,9E+09]];

    PERS robtarget H_CAM_1:=[[98.1522,-58.89,-108.72],[0.766483,-0.505835,0.353281,-0.178403],[-1,1,-2,0],[9E+09,-4.99998,46.581,9E+09,9E+09,9E+09]];
	PERS robtarget H_CAM_2:=[[98.1522,-45.58,-135.58],[0.770116,-0.507654,0.34531,-0.173119],[-1,1,-3,0],[9E+09,-4.99998,46.5812,9E+09,9E+09,9E+09]];
	PERS robtarget H_CAM_3:=[[98.1522,-39.98,-142.01],[0.807219,-0.385353,0.327992,-0.303844],[-1,1,-3,0],[9E+09,12,57.9999,9E+09,9E+09,9E+09]];
	PERS robtarget H_CAM_4:=[[98.1522,-20.35,-148.53],[0.826748,-0.369444,0.308178,-0.291592],[-1,1,-2,0],[9E+09,14,60.0001,9E+09,9E+09,9E+09]];
	PERS robtarget H_CAM_5:=[[98.1522,-10.85,-155.43],[0.769559,-0.521665,0.3083,-0.201484],[-1,1,-2,0],[9E+09,-2.00001,49.9997,9E+09,9E+09,9E+09]];
	PERS robtarget H_CAM_6:=[[98.1522,-14.24,-165.89],[0.659308,-0.625452,0.388751,-0.151641],[-1,1,-2,0],[9E+09,-15,55,9E+09,9E+09,9E+09]];
	PERS robtarget H_CAM_7:=[[98.1522,-15.81,-182.09],[0.670223,-0.62256,0.363504,-0.176309],[-1,1,-2,0],[9E+09,-18,54.9997,9E+09,9E+09,9E+09]];
	PERS robtarget H_CAM_8:=[[98.1522,-3.58,-188.22],[0.796417,-0.486379,0.272771,-0.23399],[-1,1,-3,0],[9E+09,3,54.9999,9E+09,9E+09,9E+09]];

   !!!!!!!!!!!!!
  	PERS robtarget GCam_SidePIV_S:=[[-109.269,-2,-107],[0.649686,-0.594019,0.328892,-0.341878],[-1,1,-2,0],[9E+09,-18.2042,49.7958,9E+09,9E+09,9E+09]];
  	PERS robtarget GCam_SidePIV_Sm:=[[-109.269,-1.99,-117.99],[0.609781,-0.625008,0.349951,-0.339215],[-1,1,-2,0],[9E+09,-18.2042,49.7958,9E+09,9E+09,9E+09]];
  	PERS robtarget GCam_SidePIV_M:=[[-109.269,-2,-140],[0.67995,-0.574742,0.347682,-0.294036],[-1,1,-2,0],[9E+09,-18.2042,49.7958,9E+09,9E+09,9E+09]];
  	PERS robtarget GCam_SidePIV_Em:=[[-109.269,-2,-150],[0.67995,-0.574742,0.347682,-0.294036],[-1,1,-2,0],[9E+09,-18.2042,49.7958,9E+09,9E+09,9E+09]];
  	PERS robtarget GCam_SidePIV_E:=[[-109.269,-0.93,-159.99],[0.618561,-0.622995,0.348237,-0.328618],[-1,1,-2,0],[9E+09,-18.2042,49.7958,9E+09,9E+09,9E+09]];

  	PERS robtarget HCam_SidePIV_S:=[[111.13,1.86,-103.81],[0.654832,-0.57131,-0.34952,0.350194],[-1,2,-3,0],[9E+09,-18.2042,-49.7958,9E+09,9E+09,9E+09]];
  	PERS robtarget HCam_SidePIV_Sm:=[[111.12,1.94,-118.00],[0.631899,-0.613902,-0.344567,0.324192],[-1,2,-3,0],[9E+09,-18.2042,-49.7957,9E+09,9E+09,9E+09]];
  	PERS robtarget HCam_SidePIV_M:=[[111.126,-2,-140],[0.649888,-0.476039,-0.592269,-0.0157843],[-1,1,-2,0],[9E+09,-18.2042,-49.7958,9E+09,9E+09,9E+09]];
  	PERS robtarget HCam_SidePIV_Em:=[[111.126,-2,-150],[0.649888,-0.476039,-0.592269,-0.0157843],[-1,1,-2,0],[9E+09,-18.2042,-49.7958,9E+09,9E+09,9E+09]];
  	PERS robtarget HCam_SidePIV_E:=[[111.13,0.73,-160.00],[0.621633,-0.627968,-0.342345,0.319418],[-1,2,-3,0],[9E+09,-18.2042,-49.7958,9E+09,9E+09,9E+09]];
   !!!!!!!!!!!!!
    PERS pose SRpivotYhelperGsideRound:=[[-0.0176163,-0.000339508,0.049202],[1,0,0,0]];
    PERS robtarget SPpivotYhelperGsideRoundE:=[[-62.04,37.71,-99.13],[0.633362,-0.31447,0.633322,-0.314428],[-1,1,-2,0],[9E+09,5.00002,95,9E+09,9E+09,9E+09]];
    PERS pose SRpivotYhelperHsideRound:=[[0.0116348,-0.255379,-0.025383],[1,0,0,0]];
    PERS robtarget SPpivotYhelperHsideRoundE:=[[62.027,46.7906,-99.2751],[0.690188,-0.153762,-0.69018,0.153784],[-1,1,-2,0],[9E+09,4.99999,-95.0001,9E+09,9E+09,9E+09]];

  	PERS robtarget GRnd_SidePIV_S:=[[-120.769,17.42,-200.71],[0.651172,-0.287913,0.621231,-0.327343],[-1,2,-2,0],[9E+09,5.00002,95,9E+09,9E+09,9E+09]];
  	PERS robtarget GRnd_SidePIV_Sm:=[[-120.769,17.04,-167.64],[0.651174,-0.287913,0.62123,-0.32734],[-1,2,-2,0],[9E+09,5.00002,94.9999,9E+09,9E+09,9E+09]];
  	PERS robtarget GRnd_SidePIV_M:=[[-120.769,17.92,-116.12],[0.651174,-0.287906,0.621235,-0.327337],[-1,2,-2,0],[9E+09,4.99999,95,9E+09,9E+09,9E+09]];
  	PERS robtarget GRnd_SidePIV_Em:=[[-120.769,21.68,-119.15],[0.595995,-0.227597,0.660565,-0.395783],[-1,2,-3,0],[9E+09,4.99999,105,9E+09,9E+09,9E+09]];
  	PERS robtarget GRnd_SidePIV_E:=[[-120.769,17.93,-116.14],[0.65117,-0.287909,0.621236,-0.327341],[-1,2,-2,0],[9E+09,4.99999,95,9E+09,9E+09,9E+09]];

  	PERS robtarget HRnd_SidePIV_S:=[[122.626,21.75,-200.18],[0.703025,-0.151182,-0.677087,0.156371],[-1,1,-2,0],[9E+09,5.00002,-95,9E+09,9E+09,9E+09]];
  	PERS robtarget HRnd_SidePIV_Sm:=[[122.626,21.76,-162.84],[0.703027,-0.151185,-0.677086,0.156368],[-1,1,-2,0],[9E+09,5,-95,9E+09,9E+09,9E+09]];
  	PERS robtarget HRnd_SidePIV_M:=[[122.626,21.76,-119.02],[0.703027,-0.151185,-0.677086,0.156368],[-1,0,-2,0],[9E+09,5,-95,9E+09,9E+09,9E+09]];
  	PERS robtarget HRnd_SidePIV_Em:=[[122.626,28.14,-119.7],[0.681892,-0.000934329,-0.675339,0.280964],[-1,1,-3,0],[9E+09,5,-105,9E+09,9E+09,9E+09]];
  	PERS robtarget HRnd_SidePIV_E:=[[122.626,21.76,-119.02],[0.703027,-0.151185,-0.677086,0.156368],[-1,0,-2,0],[9E+09,5,-95,9E+09,9E+09,9E+09]];
   !!!!!!!!!!!!!!!!!

    PERS robtarget OSPiv2Fwrap_G1:=[[-80.79,-4.98,-182.07],[0.670284,-0.189714,-0.414913,-0.585299],[-1,0,-2,0],[9E+09,21,-0.000317801,9E+09,9E+09,9E+09]];
 	PERS robtarget OSPiv2Fwrap_G2:=[[-91.28,-4.97,-183.63],[0.691634,-0.118244,-0.458469,-0.545405],[-1,0,-3,0],[9E+09,21,-0.000385043,9E+09,9E+09,9E+09]];
  	PERS robtarget OSPiv2Fwrap_G3:=[[-70.80,-3.90,-181.20],[0.644263,-0.288527,-0.274447,-0.652959],[-1,0,-2,0],[9E+09,21,0.00266323,9E+09,9E+09,9E+09]];
  	PERS robtarget OSPiv2Fwrap_G4:=[[0,-3.9,-181.2],[0.644265,-0.28853,-0.274445,-0.652957],[-1,0,-2,0],[9E+09,21,0.00266323,9E+09,9E+09,9E+09]];

 	PERS robtarget OSPiv2Fwrap_H1:=[[80.80,-4.99,-183.81],[0.622109,-0.376532,-0.282896,-0.625439],[-1,0,-2,0],[9E+09,21,0.00302185,9E+09,9E+09,9E+09]];
  	PERS robtarget OSPiv2Fwrap_H2:=[[88.04,-6.32,-185.36],[0.544352,-0.492096,-0.199997,-0.649248],[-1,0,-2,0],[9E+09,21,0.00317875,9E+09,9E+09,9E+09]];
  	PERS robtarget OSPiv2Fwrap_H3:=[[70,-3.88,-182.51],[0.64426,-0.288526,-0.274448,-0.652962],[-1,0,-2,0],[9E+09,21,0.0026184,9E+09,9E+09,9E+09]];
  	PERS robtarget OSPiv2Fwrap_H4:=[[0,-3.88,-182.51],[0.644261,-0.288527,-0.274448,-0.652961],[-1,0,-2,0],[9E+09,21,0.0026184,9E+09,9E+09,9E+09]];

    PERS robtarget SP_Piv0ut_GXs:=[[-31.8,-16.55,-269.25],[0.698471,-0.698472,-0.11017,-0.11017],[-1,0,-2,0],[9E+09,11.5,0,9E+09,9E+09,9E+09]];
 	PERS robtarget SP_Piv0ut_GXe:=[[-81.8,-16.55,-269.25],[0.698471,-0.698472,-0.11017,-0.11017],[-1,0,-2,0],[9E+09,11.5,0,9E+09,9E+09,9E+09]];
    PERS robtarget SP_Piv0ut_HXs:=[[31.8,-16.55,-269.25],[0.705654,-0.705654,-0.0453012,-0.0453012],[-1,1,-2,0],[9E+09,11.5,0,9E+09,9E+09,9E+09]];
    PERS robtarget SP_Piv0ut_HXe:=[[81.8,-16.55,-269.25],[0.705654,-0.705654,-0.0453012,-0.0453012],[-1,1,-2,0],[9E+09,11.5,0,9E+09,9E+09,9E+09]];
    PERS robtarget SP_Piv0ut_Ys:=[[104.208,68.5,960.7],[0.979027,2.38601E-07,5.01456E-08,-0.203733],[-1,2,-4,0],[9E+09,21,0,9E+09,9E+09,9E+09]];
    PERS robtarget SP_Piv0ut_Ye:=[[104.208,13.5,960.7],[0.979027,2.38601E-07,5.01456E-08,-0.203733],[-1,2,-4,0],[9E+09,21,0,9E+09,9E+09,9E+09]];
    PERS robtarget SP_Piv0ut_Zs:=[[104.208,36,994.2],[0.680616,-0.680616,0.191734,0.191734],[-1,1,-2,0],[9E+09,21,0,9E+09,9E+09,9E+09]];
    PERS robtarget SP_Piv0ut_Ze:=[[104.208,36,944.2],[0.680616,-0.680616,0.191734,0.191734],[-1,1,-2,0],[9E+09,21,0,9E+09,9E+09,9E+09]];

!!!!!!!!!!!!!!!!!!!!!!!!!!!!!!!!!!!!!!!!!!!!!!added 03-19-18!!!!!!!!!!!!!!!!!!!!!!!!!!!!!!!!!!!!!!!!
    PERS robtarget SP_YPIVadj_e:=[[0.86,2.59,-78.86],[0.69905,-0.106585,-0.106578,-0.699006],[-1,0,-2,0],[9E+09,21,8.56463E-05,9E+09,9E+09,9E+09]];
    PERS robtarget SP_ZPIVadj_e:=[[-17.01,-7.87,-179.30],[0.669714,-0.669689,-0.226944,-0.226928],[-1,1,-2,0],[9E+09,21,0.00064599,9E+09,9E+09,9E+09]];
    PERS pose SR_YPIVadj:=[[-0.033515,-0.692593,0.000984192],[1,0,0,0]];
    PERS pose SR_ZPIVadj:=[[-0.00343895,-0.541453,-1.49567],[1,0,0,0]];
!!!!!!!!!!!!!!!!!!!!!!!!!!!!!!!!!!!!!!!!!!!!!!!!!!!!!!!!!!!!!!!!!!!!!!!!!!!!!!!!!!!!!!!!!!!!!!!!!!!!!
!!!!!!!!!!!!!!!!!!!!!!!!!!!!!!!!!!!!!!!!!!!!!!!!!!!!!!!!!!!!!!!!!!!!!!!!!!!!!!!!!!!!!!!!!!!!!!!!!!!!!!!!!!!!!!!!!!!
!!        PJ = Pivot Joint   these are for the round shaped pivots
 	PERS robtarget G_PJRnd_1st_s:=[[-116.221,-56.77,-124],[0.71687,-0.11073,-0.684807,-0.0698286],[-1,-2,0,1],[9E+09,5,-90,9E+09,9E+09,9E+09]];
 	PERS robtarget G_PJRnd_1st_sm:=[[-116.221,-46.92,-125.74],[0.71687,-0.11073,-0.684807,-0.0698286],[-1,-2,0,1],[9E+09,5,-90,9E+09,9E+09,9E+09]];
 	PERS robtarget G_PJRnd_1st_em:=[[-116.221,6.76,-136.16],[0.731336,-0.185377,-0.643337,-0.129998],[-1,-2,0,1],[9E+09,5,-90,9E+09,9E+09,9E+09]];
 	PERS robtarget G_PJRnd_1st_e:=[[-116.221,16.76,-137],[0.744449,-0.19541,-0.62012,-0.151862],[-1,-2,0,1],[9E+09,5,-90,9E+09,9E+09,9E+09]];

 	PERS robtarget G_PJRnd_2nd_s:=[[-116.221,-56.77,-124],[0.71687,-0.110731,-0.684806,-0.0698332],[-1,-2,0,1],[9E+09,4.99997,-84.9999,9E+09,9E+09,9E+09]];
 	PERS robtarget G_PJRnd_2nd_sm:=[[-116.221,-46.92,-125.74],[0.71687,-0.11073,-0.684807,-0.0698286],[-1,-2,0,1],[9E+09,5,-85,9E+09,9E+09,9E+09]];
 	PERS robtarget G_PJRnd_2nd_em:=[[-116.221,6.76,-136.16],[0.756184,-0.180674,-0.614904,-0.132046],[-1,-2,0,1],[9E+09,4.99768,-85,9E+09,9E+09,9E+09]];
 	PERS robtarget G_PJRnd_2nd_e:=[[-116.221,16.76,-137],[0.761618,-0.196052,-0.599226,-0.149766],[-1,-2,0,1],[9E+09,4.99767,-74.9999,9E+09,9E+09,9E+09]];

 	PERS robtarget G_PJRnd_3rd_s:=[[-116.221,-56.77,-124],[0.71687,-0.11073,-0.684807,-0.0698286],[-1,-2,0,1],[9E+09,5,-85,9E+09,9E+09,9E+09]];
 	PERS robtarget G_PJRnd_3rd_sm:=[[-116.221,-46.92,-125.74],[0.71687,-0.11073,-0.684807,-0.0698286],[-1,-2,0,1],[9E+09,5,-85,9E+09,9E+09,9E+09]];
 	PERS robtarget G_PJRnd_3rd_em:=[[-116.221,6.76,-136.16],[0.759108,-0.156585,-0.621504,-0.11388],[-1,-2,0,1],[9E+09,5,-85,9E+09,9E+09,9E+09]];
 	PERS robtarget G_PJRnd_3rd_e:=[[-116.221,16.76,-137],[0.690713,-0.364323,-0.609662,-0.136004],[-1,-2,1,1],[9E+09,5,-85,9E+09,9E+09,9E+09]];

 	PERS robtarget G_PJRnd_4th_s:=[[-116.221,-56.77,-124],[0.71687,-0.11073,-0.684807,-0.0698286],[-1,-2,0,1],[9E+09,5,-85,9E+09,9E+09,9E+09]];
 	PERS robtarget G_PJRnd_4th_sm:=[[-116.221,-46.92,-125.74],[0.71687,-0.11073,-0.684807,-0.0698286],[-1,-2,0,1],[9E+09,5,-85,9E+09,9E+09,9E+09]];
 	PERS robtarget G_PJRnd_4th_em:=[[-116.221,6.76,-136.16],[0.759108,-0.156585,-0.621504,-0.11388],[-1,-2,0,1],[9E+09,5,-85,9E+09,9E+09,9E+09]];
 	PERS robtarget G_PJRnd_4th_e:=[[-116.221,16.76,-137],[0.690713,-0.364323,-0.609662,-0.136004],[-1,-2,1,1],[9E+09,5,-85,9E+09,9E+09,9E+09]];

 	PERS robtarget H_PJRnd_1st_s:=[[116.85,-50.63,-124.76],[0.645351,-0.379915,0.599982,-0.28144],[-1,1,2,0],[9E+09,4.99999,90.0002,9E+09,9E+09,9E+09]];
 	PERS robtarget H_PJRnd_1st_sm:=[[116.84,-40.53,-125.74],[0.633823,-0.410174,0.57585,-0.313723],[-1,1,2,0],[9E+09,4.99999,90.0001,9E+09,9E+09,9E+09]];
 	PERS robtarget H_PJRnd_1st_em:=[[116.84,-1.05,-133.41],[0.656479,-0.48509,0.443945,-0.369643],[-1,1,2,0],[9E+09,4.99999,90,9E+09,9E+09,9E+09]];
 	PERS robtarget H_PJRnd_1st_e:=[[116.85,12.27,-135.78],[0.684689,-0.478579,0.414268,-0.361309],[-1,1,1,0],[9E+09,4.99999,90,9E+09,9E+09,9E+09]];

 	PERS robtarget H_PJRnd_2nd_s:=[[116.84,-52.58,-123.26],[0.668155,-0.357654,0.579241,-0.300222],[-1,1,2,0],[9E+09,4.99999,84.9999,9E+09,9E+09,9E+09]];
 	PERS robtarget H_PJRnd_2nd_sm:=[[116.86,-41.60,-125.09],[0.668503,-0.394742,0.522148,-0.35305],[-1,1,2,0],[9E+09,5.00003,85,9E+09,9E+09,9E+09]];
 	PERS robtarget H_PJRnd_2nd_em:=[[116.848,0.57,-132.97],[0.690657,-0.443246,0.412829,-0.395092],[-1,1,1,0],[9E+09,4.99997,84.9999,9E+09,9E+09,9E+09]];
 	PERS robtarget H_PJRnd_2nd_e:=[[117.21,10.44,-135.86],[0.701835,-0.479653,0.380667,-0.36394],[-1,1,1,0],[9E+09,4.99997,75,9E+09,9E+09,9E+09]];

 	PERS robtarget H_PJRnd_3rd_s:=[[116.848,-56.77,-124],[0.645356,-0.379913,0.59998,-0.281436],[-1,1,2,0],[9E+09,5,85,9E+09,9E+09,9E+09]];
 	PERS robtarget H_PJRnd_3rd_sm:=[[116.848,-46.92,-125.74],[0.625682,-0.424599,0.565304,-0.32965],[-1,1,2,0],[9E+09,5,85,9E+09,9E+09,9E+09]];
 	PERS robtarget H_PJRnd_3rd_em:=[[116.848,6.76,-136.16],[0.653344,-0.494982,0.443626,-0.362395],[-1,1,2,0],[9E+09,5,85,9E+09,9E+09,9E+09]];
 	PERS robtarget H_PJRnd_3rd_e:=[[116.848,16.76,-137],[0.681465,-0.518041,0.399083,-0.32859],[-1,1,2,0],[9E+09,5,85,9E+09,9E+09,9E+09]];

 	PERS robtarget H_PJRnd_4th_s:=[[112.848,-56.77,-124],[0.645356,-0.379913,0.59998,-0.281436],[-1,1,2,0],[9E+09,5,85,9E+09,9E+09,9E+09]];
 	PERS robtarget H_PJRnd_4th_sm:=[[112.848,-46.92,-125.74],[0.625682,-0.424599,0.565304,-0.32965],[-1,1,2,0],[9E+09,5,85,9E+09,9E+09,9E+09]];
 	PERS robtarget H_PJRnd_4th_em:=[[112.848,6.76,-136.16],[0.653344,-0.494982,0.443626,-0.362395],[-1,1,2,0],[9E+09,5,85,9E+09,9E+09,9E+09]];
 	PERS robtarget H_PJRnd_4th_e:=[[110.848,16.76,-137],[0.681465,-0.518041,0.399083,-0.32859],[-1,1,2,0],[9E+09,5,85,9E+09,9E+09,9E+09]];

!!!!!!!!!!!!!!!!!!!!!!!!!!!!!!!!!!!!!!!!!!!!!!!!!!!!!!!!!!!!!!!!!!!!!!!!!!!!!!!!!!!!!!!!!!!!!!!!!!!!!!!!!!!!!!!!!!!!!!!!!!!!!!!!!
!!        PJ = Pivot Joint   these are for the CAM shaped pivots
 	PERS robtarget H_PJCam_1st_s:=[[110.602,-2.4,-110.82],[0.398951,-0.65704,-0.250921,0.588367],[-1,-3,3,1],[9E+09,4.67604E-05,-90.0002,9E+09,9E+09,9E+09]];
	PERS robtarget H_PJCam_1st_sm:=[[110.602,-5.8,-110.15],[0.318277,-0.633541,-0.321425,0.627703],[-1,-4,3,1],[9E+09,-4.98748E-06,-90,9E+09,9E+09,9E+09]];
	PERS robtarget H_PJCam_1st_em:=[[110.602,-44.04,-99.16],[0.309721,-0.615411,-0.329677,0.645488],[-1,-4,3,1],[9E+09,5.73674E-05,-90.0003,9E+09,9E+09,9E+09]];
	PERS robtarget H_PJCam_1st_e:=[[110.602,-51.33,-96.68],[0.301369,-0.599085,-0.337318,0.660675],[-1,-4,3,1],[9E+09,3.65824E-05,-90.0001,9E+09,9E+09,9E+09]];

	PERS robtarget H_PJCam_2nd_s:=[[110.602,-1,-111.55],[0.398955,-0.657033,-0.250926,0.58837],[-1,-3,3,1],[9E+09,5,-90,9E+09,9E+09,9E+09]];
	PERS robtarget H_PJCam_2nd_sm:=[[110.602,-5.79,-110.26],[0.318281,-0.633538,-0.321426,0.627704],[-1,-4,3,1],[9E+09,5,-90,9E+09,9E+09,9E+09]];
	PERS robtarget H_PJCam_2nd_em:=[[110.602,-45.58,-99.59],[0.309717,-0.615414,-0.32968,0.645486],[-1,-4,3,1],[9E+09,5,-90,9E+09,9E+09,9E+09]];
    PERS robtarget H_PJCam_2nd_e:=[[110.602,-50.41,-98.3],[0.306036,-0.582148,-0.33034,0.676994],[-1,-4,3,1],[9E+09,5,-90,9E+09,9E+09,9E+09]];

 	PERS robtarget H_PJCam_3rd_s:=[[110.602,-1,-111.55],[0.398955,-0.657033,-0.250926,0.58837],[-1,-3,3,1],[9E+09,5,-90,9E+09,9E+09,9E+09]];
	PERS robtarget H_PJCam_3rd_sm:=[[110.602,-5.79,-110.26],[0.318281,-0.633538,-0.321426,0.627704],[-1,-4,3,1],[9E+09,5,-90,9E+09,9E+09,9E+09]];
	PERS robtarget H_PJCam_3rd_em:=[[110.602,-45.58,-99.59],[0.309717,-0.615414,-0.32968,0.645486],[-1,-4,3,1],[9E+09,5,-90,9E+09,9E+09,9E+09]];
    PERS robtarget H_PJCam_3rd_e:=[[110.602,-50.41,-98.3],[0.306036,-0.582148,-0.33034,0.676994],[-1,-4,3,1],[9E+09,5,-90,9E+09,9E+09,9E+09]];

	PERS robtarget H_PJCam_4th_s:=[[110.602,-1.71,-111.68],[0.42228,-0.640978,-0.232213,0.597415],[-1,-3,3,1],[9E+09,2.59754E-05,-90,9E+09,9E+09,9E+09]];
	PERS robtarget H_PJCam_4th_sm:=[[110.602,-7.26,-110.35],[0.358651,-0.636258,-0.280366,0.622848],[-1,-4,3,1],[9E+09,-5.20202E-06,-90,9E+09,9E+09,9E+09]];
	PERS robtarget H_PJCam_4th_em:=[[110.602,-46.66,-100.15],[0.343263,-0.630093,-0.29504,0.630955],[-1,-4,3,1],[9E+09,2.59754E-05,-89.9999,9E+09,9E+09,9E+09]];
    PERS robtarget H_PJCam_4th_e:=[[110.602,-55.59,-97.87],[0.348944,-0.623408,-0.28586,0.638659],[-1,-4,3,1],[9E+09,-4.67719E-05,-90,9E+09,9E+09,9E+09]];

	PERS robtarget H_PJCam_5th_s:=[[110.602,-6.5,-156.6],[0.39895,-0.657033,-0.250928,0.588372],[-1,-3,3,1],[9E+09,5,-90,9E+09,9E+09,9E+09]];
	PERS robtarget H_PJCam_5th_sm:=[[110.602,-11.35,-154.75],[0.318286,-0.633538,-0.321426,0.627702],[-1,-4,3,1],[9E+09,5,-90,9E+09,9E+09,9E+09]];
	PERS robtarget H_PJCam_5th_em:=[[110.602,-67.65,-139.8],[0.309714,-0.615412,-0.329681,0.645489],[-1,-4,3,1],[9E+09,5,-90,9E+09,9E+09,9E+09]];
	PERS robtarget H_PJCam_5th_e:=[[110.602,-72.5,-138.5],[0.306033,-0.58215,-0.330337,0.676995],[-1,-4,3,1],[9E+09,5,-90,9E+09,9E+09,9E+09]];

 	PERS robtarget G_PJCam_1st_s:=[[-107.775,-5.82,-110.51],[0.664139,-0.454628,0.507295,-0.308033],[-1,1,-2,0],[9E+09,-0.000171267,90.0005,9E+09,9E+09,9E+09]];
	PERS robtarget G_PJCam_1st_sm:=[[-107.775,-9.93,-108.79],[0.599292,-0.389593,0.57554,-0.397266],[-1,1,-2,0],[9E+09,-4.98748E-06,89.9999,9E+09,9E+09,9E+09]];
	PERS robtarget G_PJCam_1st_em:=[[-107.775,-47.4,-97.95],[0.58619,-0.377085,0.588845,-0.409206],[-1,1,-2,0],[9E+09,2.59754E-05,90.0001,9E+09,9E+09,9E+09]];
    PERS robtarget G_PJCam_1st_e:=[[-107.775,-52.34,-97.4],[0.585528,-0.365611,0.587357,-0.422489],[-1,1,-2,0],[9E+09,-4.67719E-05,89.9999,9E+09,9E+09,9E+09]];

	PERS robtarget G_PJCam_2nd_s:=[[-107.775,-1,-111.55],[0.664146,-0.454653,0.507271,-0.30802],[-1,1,-2,0],[9E+09,5,90,9E+09,9E+09,9E+09]];
	PERS robtarget G_PJCam_2nd_sm:=[[-107.775,-5.79,-110.26],[0.606546,-0.394607,0.567886,-0.392291],[-1,1,-2,0],[9E+09,5,90,9E+09,9E+09,9E+09]];
	PERS robtarget G_PJCam_2nd_em:=[[-107.775,-45.58,-99.59],[0.599356,-0.386244,0.575437,-0.400574],[-1,1,-2,0],[9E+09,5,90,9E+09,9E+09,9E+09]];
	PERS robtarget G_PJCam_2nd_e:=[[-107.775,-50.41,-98.3],[0.585534,-0.365613,0.58735,-0.422489],[-1,1,-2,0],[9E+09,5,90,9E+09,9E+09,9E+09]];

 	PERS robtarget G_PJCam_3rd_s:=[[-107.775,-1,-111.55],[0.664146,-0.454653,0.507271,-0.30802],[-1,1,-2,0],[9E+09,5,90,9E+09,9E+09,9E+09]];
	PERS robtarget G_PJCam_3rd_sm:=[[-107.775,-5.79,-110.26],[0.606546,-0.394607,0.567886,-0.392291],[-1,1,-2,0],[9E+09,5,90,9E+09,9E+09,9E+09]];
	PERS robtarget G_PJCam_3rd_em:=[[-107.775,-45.58,-99.59],[0.599356,-0.386244,0.575437,-0.400574],[-1,1,-2,0],[9E+09,5,90,9E+09,9E+09,9E+09]];
    PERS robtarget G_PJCam_3rd_e:=[[-107.775,-50.41,-98.3],[0.585534,-0.365613,0.58735,-0.422489],[-1,1,-2,0],[9E+09,5,90,9E+09,9E+09,9E+09]];

	PERS robtarget G_PJCam_4th_s:=[[-107.775,-4.09,-111.57],[0.668527,-0.451948,0.50314,-0.309297],[-1,1,-2,0],[9E+09,-0.000399902,89.9987,9E+09,9E+09,9E+09]];
	PERS robtarget G_PJCam_4th_sm:=[[-107.775,-9.52,-111.1],[0.610875,-0.406949,0.562731,-0.380207],[-1,1,-2,0],[9E+09,-5.69499E-05,89.9997,9E+09,9E+09,9E+09]];
	PERS robtarget G_PJCam_4th_em:=[[-107.775,-47.67,-100.86],[0.60677,-0.402434,0.567094,-0.385073],[-1,1,-2,0],[9E+09,-5.69499E-05,89.9998,9E+09,9E+09,9E+09]];
	PERS robtarget G_PJCam_4th_e:=[[-107.775,-57.31,-99.48],[0.597922,-0.371998,0.574618,-0.417038],[-1,1,-3,0],[9E+09,-4.98748E-06,89.9999,9E+09,9E+09,9E+09]];

	PERS robtarget G_PJCam_5th_s:=[[-107.775,-6.5,-156.6],[0.664146,-0.454652,0.507271,-0.308022],[-1,1,-2,0],[9E+09,5,90,9E+09,9E+09,9E+09]];
	PERS robtarget G_PJCam_5th_sm:=[[-107.775,-11.35,-154.75],[0.606547,-0.39461,0.567882,-0.392293],[-1,1,-2,0],[9E+09,5,90,9E+09,9E+09,9E+09]];
	PERS robtarget G_PJCam_5th_em:=[[-107.775,-67.65,-139.8],[0.599352,-0.386244,0.575442,-0.400573],[-1,1,-2,0],[9E+09,5,90,9E+09,9E+09,9E+09]];
	PERS robtarget G_PJCam_5th_e:=[[-107.775,-72.5,-138.5],[0.615886,-0.387535,0.555435,-0.402483],[-1,1,-2,0],[9E+09,5,90,9E+09,9E+09,9E+09]];


    !!!!!!!!!!!!!!!!!!!!!!!!!!!!!!!!!!!!!!!!!!!!!!!!!!!!!!!!!!!!!!!!!!!!!!!!!!!!!!!!!!!!!!!!!!!!!!!!!!!!!!!!!!!!!!!!!!!!!!!!!!!!!
    !!!    SEARCHES FOR G/H PIV 1 THRU 8
    !!!!!!!!!!!!!!!!!!!!!!!!!!!!!!!!!!!!!!!!!!!!!!!!!!!!!!!!!!!!!!!!!!!!!!!!!!!!!!!!!!!!!!!!!!!!!!!!!!!!!!!!!!!!!!!!!!!!!!!!!!
  !!        18 = points 1 thru 8, in CAM or RND Pivots
    PERS robtarget SP_gPivRnd_18_Xs:=[[-158.8,-16.55,-269.25],[0.074768,-0.0747681,-0.703143,-0.703143],[-1,0,-3,0],[9E+09,8.5359,48.4641,9E+09,9E+09,9E+09]];
 	PERS robtarget SP_gPivRnd_18_Xe:=[[-108.8,-16.55,-269.25],[0.074768,-0.0747681,-0.703143,-0.703143],[-1,0,-3,0],[9E+09,8.5359,48.4641,9E+09,9E+09,9E+09]];
 	PERS robtarget SP_hPivRnd_18_Xs:=[[158.8,-16.55,-269.25],[0.6019,-0.601901,-0.371101,-0.3711],[-1,0,-1,0],[9E+09,8.5359,-48.4641,9E+09,9E+09,9E+09]];
 	PERS robtarget SP_hPivRnd_18_Xe:=[[108.8,-16.55,-269.25],[0.6019,-0.601901,-0.371101,-0.3711],[-1,0,-1,0],[9E+09,8.5359,-48.4641,9E+09,9E+09,9E+09]];

    PERS robtarget SP_gPivCam_18_Xs:=[[-31.8,-16.55,-269.25],[0.669176,-0.669177,-0.228479,-0.228479],[-1,0,-1,0],[9E+09,0,-45,9E+09,9E+09,9E+09]];
 	PERS robtarget SP_gPivCam_18_Xe:=[[-81.8,-16.55,-269.25],[0.669176,-0.669177,-0.228479,-0.228479],[-1,0,-1,0],[9E+09,0,-45,9E+09,9E+09,9E+09]];
 	PERS robtarget SP_hPivCam_18_Xs:=[[31.8,-16.55,-269.25],[0.228057,-0.228057,-0.669321,-0.66932],[-1,0,-3,0],[9E+09,0,45,9E+09,9E+09,9E+09]];
 	PERS robtarget SP_hPivCam_18_Xe:=[[81.8,-16.55,-269.25],[0.228057,-0.228057,-0.669321,-0.66932],[-1,0,-3,0],[9E+09,0,45,9E+09,9E+09,9E+09]];

 	PERS robtarget SP_HPivRND_18_Ys:=[[134.755,63.5,811.2],[7.62829E-08,-0.962536,0.271153,1.37778E-07],[-1,1,-2,0],[9E+09,8.5359,-48.4641,9E+09,9E+09,9E+09]];
 	PERS robtarget SP_HPivRND_18_Ye:=[[134.755,13.5,811.2],[7.62829E-08,-0.962536,0.271153,1.37778E-07],[-1,1,-2,0],[9E+09,8.5359,-48.4641,9E+09,9E+09,9E+09]];
 	PERS robtarget SP_HPivRND_18_Zs:=[[134.755,25,977.2],[0.680616,-0.680616,0.191734,0.191734],[-1,-1,0,0],[9E+09,8.5359,-48.4641,9E+09,9E+09,9E+09]];
 	PERS robtarget SP_HPivRND_18_Ze:=[[134.755,25,942.2],[0.680616,-0.680616,0.191734,0.191734],[-1,-1,0,0],[9E+09,8.5359,-48.4641,9E+09,9E+09,9E+09]];

 	PERS robtarget SP_GPivRND_18_Ys:=[[-133.168,63.5,833.7],[3.37488E-07,0.324654,-0.945833,3.78335E-08],[-1,0,0,0],[9E+09,8.5359,48.4641,9E+09,9E+09,9E+09]];
 	PERS robtarget SP_GPivRND_18_Ye:=[[-133.168,13.5,833.7],[3.37488E-07,0.324654,-0.945833,3.78335E-08],[-1,0,0,0],[9E+09,8.5359,48.4641,9E+09,9E+09,9E+09]];
 	PERS robtarget SP_GPivRND_18_Zs:=[[-133.168,25,977.2],[0.229565,-0.229565,0.668805,0.668805],[0,-1,2,0],[9E+09,8.5359,48.4641,9E+09,9E+09,9E+09]];
 	PERS robtarget SP_GPivRND_18_Ze:=[[-133.168,25,942.2],[0.229565,-0.229565,0.668805,0.668805],[0,-1,2,0],[9E+09,8.5359,48.4641,9E+09,9E+09,9E+09]];

  	PERS robtarget SP_HPivCAM_18_Ys:=[[108.152,63.5,826.2],[7.62829E-08,-0.962536,0.271153,1.37778E-07],[-1,1,-2,0],[9E+09,0,45,9E+09,9E+09,9E+09]];
 	PERS robtarget SP_HPivCAM_18_Ye:=[[108.152,13.5,826.2],[7.62829E-08,-0.962536,0.271153,1.37778E-07],[-1,1,-2,0],[9E+09,0,45,9E+09,9E+09,9E+09]];
 	PERS robtarget SP_HPivCAM_18_Zs:=[[108.152,25,977.2],[0.646945,-0.646944,0.285416,0.285418],[-1,2,-2,0],[9E+09,0,45,9E+09,9E+09,9E+09]];
 	PERS robtarget SP_HPivCAM_18_Ze:=[[108.152,25,942.2],[0.646944,-0.646947,0.285414,0.285417],[-1,2,-2,0],[9E+09,0,45,9E+09,9E+09,9E+09]];

 	PERS robtarget SP_GPivCAM_18_Ys:=[[-98.072,63.5,953.7],[0.918423,-1.83184E-08,6.48462E-09,0.3956],[-1,0,-1,1],[9E+09,0,-45,9E+09,9E+09,9E+09]];
 	PERS robtarget SP_GPivCAM_18_Ye:=[[-98.072,13.5,953.7],[0.918423,-1.83184E-08,6.48462E-09,0.3956],[-1,0,-1,1],[9E+09,0,-45,9E+09,9E+09,9E+09]];
 	PERS robtarget SP_GPivCAM_18_Zs:=[[-98.072,25,977.2],[0.703252,-0.703252,-0.0737343,-0.0737346],[-1,0,-1,0],[9E+09,0,-45,9E+09,9E+09,9E+09]];
 	PERS robtarget SP_GPivCAM_18_Ze:=[[-98.072,25,942.2],[0.703252,-0.703252,-0.0737343,-0.0737346],[-1,0,-1,0],[9E+09,0,-45,9E+09,9E+09,9E+09]];

    !!!!!!!!!!!!!!!!!!!!!!!!!!!!!!!!!!!!!!!!!!!!!!!!!!!!!!!!!!!!!!!!!!!!!!!!!!!!!!!!!!!!!!!!!!!!!!!!!!!!!!!!!!!!!!!!!!!!!!!!!!!!!
    !!!    SEARCHES FOR G/H           PJ = PIVOT JOINT            !!!
    !!!!!!!!!!!!!!!!!!!!!!!!!!!!!!!!!!!!!!!!!!!!!!!!!!!!!!!!!!!!!!!!!!!!!!!!!!!!!!!!!!!!!!!!!!!!!!!!!!!!!!!!!!!!!!!!!!!!!!!!!!

    PERS robtarget SP_gPivRnd_PJ_Xs:=[[-19.8,-16.55,-269.25],[0.671032,-0.741422,0.00221101,0.00200072],[-1,0,-1,0],[9E+09,5,-60,9E+09,9E+09,9E+09]];
 	PERS robtarget SP_gPivRnd_PJ_Xe:=[[-69.8,-16.55,-269.25],[0.671032,-0.741422,0.00221101,0.00200072],[-1,0,-1,0],[9E+09,5,-60,9E+09,9E+09,9E+09]];
 	PERS robtarget SP_hPivRnd_PJ_Xs:=[[19.8,-16.55,-269.25],[0.0441236,-0.0785833,-0.868404,-0.487598],[-1,1,0,0],[9E+09,5,90,9E+09,9E+09,9E+09]];
 	PERS robtarget SP_hPivRnd_PJ_Xe:=[[69.8,-16.55,-269.25],[0.0441236,-0.0785833,-0.868404,-0.487598],[-1,1,0,0],[9E+09,5,90,9E+09,9E+09,9E+09]];

    PERS robtarget SP_gPivCam_PJ_Xs:=[[-170.8,-16.55,-269.25],[0.0596632,-0.110181,-0.872423,-0.472418],[-1,-2,-2,1],[9E+09,0,90,9E+09,9E+09,9E+09]];
 	PERS robtarget SP_gPivCam_PJ_Xe:=[[-120.8,-16.55,-269.25],[0.0596632,-0.110181,-0.872423,-0.472418],[-1,-2,-2,1],[9E+09,0,90,9E+09,9E+09,9E+09]];
 	PERS robtarget SP_hPivCam_PJ_Xs:=[[170.8,-16.55,-269.25],[0.981346,-0.071223,0.0129263,0.1781],[0,-1,-1,0],[9E+09,0,-90,9E+09,9E+09,9E+09]];
 	PERS robtarget SP_hPivCam_PJ_Xe:=[[120.8,-16.55,-269.25],[0.981346,-0.071223,0.0129263,0.1781],[0,-1,-1,0],[9E+09,0,-90,9E+09,9E+09,9E+09]];

 	PERS robtarget SP_HPivRND_PJ_Ys:=[[132.848,63.5,811.2],[1.18971E-07,-0.582357,0.812933,2.40784E-08],[-1,1,-1,0],[9E+09,5,90,9E+09,9E+09,9E+09]];
 	PERS robtarget SP_HPivRND_PJ_Ye:=[[132.848,13.5,811.2],[1.18971E-07,-0.582357,0.812933,2.40784E-08],[-1,1,-1,0],[9E+09,5,90,9E+09,9E+09,9E+09]];
 	PERS robtarget SP_HPivRND_PJ_Zs:=[[132.848,25,977.2],[0.0637268,-0.0637268,-0.704229,-0.704229],[-1,1,0,0],[9E+09,5,90,9E+09,9E+09,9E+09]];
 	PERS robtarget SP_HPivRND_PJ_Ze:=[[132.848,25,942.2],[0.0637268,-0.0637268,-0.704229,-0.704229],[-1,1,0,0],[9E+09,5,90,9E+09,9E+09,9E+09]];

 	PERS robtarget SP_GPivRND_PJ_Ys:=[[-132.221,63.5,833.7],[6.61632E-09,0.955297,0.295649,-1.24719E-08],[-1,1,-1,0],[9E+09,5,-90,9E+09,9E+09,9E+09]];
 	PERS robtarget SP_GPivRND_PJ_Ye:=[[-132.221,13.5,833.7],[6.61632E-09,0.955297,0.295649,-1.24719E-08],[-1,1,-1,0],[9E+09,5,-90,9E+09,9E+09,9E+09]];
 	PERS robtarget SP_GPivRND_PJ_Zs:=[[-132.221,-95,977.2],[0.695296,0.695296,0.128698,-0.128698],[-1,2,-1,0],[9E+09,5,-90,9E+09,9E+09,9E+09]];
 	PERS robtarget SP_GPivRND_PJ_Ze:=[[-132.221,-95,942.2],[0.695296,0.695296,0.128698,-0.128698],[-1,2,-1,0],[9E+09,5,-90,9E+09,9E+09,9E+09]];

  	PERS robtarget SP_HPivCAM_PJ_Ys:=[[100.602,63.5,962.45],[0.977308,-1.46315E-09,3.11534E-08,0.211823],[-1,-2,-1,0],[9E+09,0,-90,9E+09,9E+09,9E+09]];
 	PERS robtarget SP_HPivCAM_PJ_Ye:=[[100.602,13.5,962.45],[0.977308,-1.46315E-09,3.11534E-08,0.211823],[-1,-2,-1,0],[9E+09,0,-90,9E+09,9E+09,9E+09]];
 	PERS robtarget SP_HPivCAM_PJ_Zs:=[[100.602,-95,977.2],[0.655082,0.655082,0.26621,-0.26621],[-1,-3,-1,0],[9E+09,0,-90,9E+09,9E+09,9E+09]];
 	PERS robtarget SP_HPivCAM_PJ_Ze:=[[100.602,-95,942.2],[0.655082,0.655082,0.26621,-0.26621],[-1,-3,-1,0],[9E+09,0,-90,9E+09,9E+09,9E+09]];

 	PERS robtarget SP_GPivCAM_PJ_Ys:=[[-97.7754,63.5,963.7],[0.125298,-1.8924E-08,-7.50359E-08,-0.992119],[-1,0,-3,1],[9E+09,0,90,9E+09,9E+09,9E+09]];
 	PERS robtarget SP_GPivCAM_PJ_Ye:=[[-97.7754,13.5,963.7],[0.125298,-1.8924E-08,-7.50359E-08,-0.992119],[-1,0,-3,1],[9E+09,0,90,9E+09,9E+09,9E+09]];
 	PERS robtarget SP_GPivCAM_PJ_Zs:=[[-97.7754,25,977.2],[0.0885989,-0.088599,-0.701534,-0.701534],[-1,-2,-2,1],[9E+09,0,90,9E+09,9E+09,9E+09]];
 	PERS robtarget SP_GPivCAM_PJ_Ze:=[[-97.7754,25,942.2],[0.0885989,-0.088599,-0.701534,-0.701534],[-1,-2,-2,1],[9E+09,0,90,9E+09,9E+09,9E+09]];

    !!!!!!!!!!!!!!!!!!!!!!!!!!!!!!!!!!!!!!!!!!!!!!!!!!!!!!!!!!!!!!!!!!!!!!!!!!!!!!!!!!!!!!!!!!!!!!!!!!!!!!!!!!!!!!!!!!!!!!!!!!!!!
    !!!    SEARCHES FOR PIVOT in 180
    !!!!!!!!!!!!!!!!!!!!!!!!!!!!!!!!!!!!!!!!!!!!!!!!!!!!!!!!!!!!!!!!!!!!!!!!!!!!!!!!!!!!!!!!!!!!!!!!!!!!!!!!!!!!!!!!!!!!!!!!!!!!!

    PERS robtarget Piv2Fwrap_RS:=[[96.91,7.59,-156.84],[0.00115525,-0.000739029,0.767298,-0.641289],[-1,1,-2,0],[9E+09,15,180,9E+09,9E+09,9E+09]];
    PERS robtarget Piv2Fwrap_RE:=[[-98.75,8.45,-156.01],[0.00114663,-0.00074178,0.767298,-0.641289],[-1,1,-2,0],[9E+09,15,180,9E+09,9E+09,9E+09]];
    PERS robtarget Piv2Fwrap_GS:=[[-106.74,12.00,-155.01],[0.000224929,0.000204849,0.721171,-0.692757],[-1,1,-2,0],[9E+09,24,180,9E+09,9E+09,9E+09]];
    PERS robtarget Piv2Fwrap_GE:=[[0,12,-155.01],[0.000224929,0.000204849,0.721171,-0.692757],[-1,1,-2,0],[9E+09,24,180,9E+09,9E+09,9E+09]];
    PERS robtarget Piv2Fwrap_HS:=[[104.60,10.24,-155.76],[0.000221724,0.000202154,0.721171,-0.692757],[-1,1,-2,0],[9E+09,24,180,9E+09,9E+09,9E+09]];
    PERS robtarget Piv2Fwrap_HE:=[[-10,12,-155.01],[0.000224929,0.000204849,0.721171,-0.692757],[-1,1,-2,0],[9E+09,24,180,9E+09,9E+09,9E+09]];

    PERS robtarget SP_PIV180_XS:=[[-179.3,-95,894.7],[0.0297707,0.0371963,0.772847,-0.632801],[-1,1,-2,0],[9E+09,24,180,9E+09,9E+09,9E+09]];
 	PERS robtarget SP_Piv180_Xe:=[[-129.3,-95,894.7],[0.0297708,0.0371963,0.772847,-0.632801],[-1,1,-2,0],[9E+09,24,180,9E+09,9E+09,9E+09]];
    PERS robtarget SP_Piv180_Ys:=[[-101.631,63.5,958.7],[0.668512,9.04063E-08,-3.35034E-08,0.743702],[-1,-2,-1,0],[9E+09,24,180,9E+09,9E+09,9E+09]];
 	PERS robtarget SP_Piv180_Ye:=[[-101.631,13.5,958.7],[0.668512,9.04063E-08,-3.35034E-08,0.743702],[-1,-2,-1,0],[9E+09,24,180,9E+09,9E+09,9E+09]];
    PERS robtarget SP_Piv180_Zs:=[[-101.631,-99.75,977.2],[0.22387,0.223869,0.670733,-0.670733],[-1,1,-2,0],[9E+09,24,180,9E+09,9E+09,9E+09]];
 	PERS robtarget SP_Piv180_Ze:=[[-101.631,-99.75,942.2],[0.22387,0.223869,0.670733,-0.670733],[-1,1,-2,0],[9E+09,24,180,9E+09,9E+09,9E+09]];

          ! SEARCES FOR G/H SIDE WELDS (USED TO BE CALLED THE 40's)
     PERS ROBTARGET  SP_HRnd_Side_XS := [[158.8,-16.55,-269.25],[0.505591,-0.828545,-0.205385,-0.125329],[-1,0,0,0],[9E+09,0,-90,9E+09,9E+09,9E+09]];
     PERS ROBTARGET  SP_HRnd_Side_XE := [[108.8,-16.55,-269.25],[0.505591,-0.828545,-0.205385,-0.125329],[-1,0,0,0],[9E+09,0,-90,9E+09,9E+09,9E+09]];
     PERS ROBTARGET  SP_HRnd_Side_YS := [[109.126,63.5,833.7],[1.45997E-08,0.971896,0.23541,-5.32529E-09],[-1,0,0,0],[9E+09,0,-90,9E+09,9E+09,9E+09]];
     PERS ROBTARGET  SP_HRnd_Side_YE := [[109.126,13.5,833.7],[1.45997E-08,0.971896,0.23541,-5.32529E-09],[-1,0,0,0],[9E+09,0,-90,9E+09,9E+09,9E+09]];
     PERS ROBTARGET  SP_HRnd_Side_ZS := [[109.126,-95,992.2],[0.687234,0.687234,0.16646,-0.16646],[-1,1,-1,0],[9E+09,0,-90,9E+09,9E+09,9E+09]];
     PERS ROBTARGET  SP_HRnd_Side_ZE := [[109.126,-95,942.2],[0.687234,0.687234,0.16646,-0.16646],[-1,1,-1,0],[9E+09,0,-90,9E+09,9E+09,9E+09]];
     !!!!!!!!!!!!!!!!!!!!!!!!!!!!!!!!!!!!!!!!!!
     PERS ROBTARGET  SP_GRnd_Side_XS := [[-158.8,-16.55,-269.25],[0.285529,-0.488698,0.711816,0.415892],[-1,0,0,0],[9E+09,0,90,9E+09,9E+09,9E+09]];
     PERS ROBTARGET  SP_GRnd_Side_XE := [[-108.8,-16.55,-269.25],[0.285529,-0.488698,0.711816,0.415892],[-1,0,0,0],[9E+09,0,90,9E+09,9E+09,9E+09]];
     PERS ROBTARGET  SP_GRnd_Side_YS := [[-107.269,63.5,833.7],[1.41006E-07,0.41919,-0.907898,-2.81481E-07],[-1,1,-1,0],[9E+09,0,90,9E+09,9E+09,9E+09]];
     PERS ROBTARGET  SP_GRnd_Side_YE := [[-107.269,13.5,833.7],[1.41006E-07,0.41919,-0.907898,-2.81481E-07],[-1,1,-1,0],[9E+09,0,90,9E+09,9E+09,9E+09]];
     PERS ROBTARGET  SP_GRnd_Side_ZS := [[-107.269,23.75,992.2],[0.203561,-0.203561,0.677172,0.677173],[-1,2,-1,0],[9E+09,0,90,9E+09,9E+09,9E+09]];
     PERS ROBTARGET  SP_GRnd_Side_ZE := [[-107.269,23.75,942.2],[0.203561,-0.203561,0.677172,0.677173],[-1,2,-1,0],[9E+09,0,90,9E+09,9E+09,9E+09]];
    !!!!!!!!!!!!!!!!!!

     PERS ROBTARGET  SP_HCam_Side_XS := [[170.8,-16.55,-269.25],[0.676221,-0.676221,-0.206699,-0.206699],[-1,0,-1,0],[9E+09,-18.2042,-49.7958,9E+09,9E+09,9E+09]];
     PERS ROBTARGET  SP_HCam_Side_XE := [[120.8,-16.55,-269.25],[0.676221,-0.676221,-0.206699,-0.206699],[-1,0,-1,0],[9E+09,-18.2042,-49.7958,9E+09,9E+09,9E+09]];
     PERS ROBTARGET  SP_HCam_Side_YS := [[102.126,63.5,833.7],[6.88078E-09,0.956321,0.292317,-1.26749E-08],[-1,0,-1,0],[9E+09,-18.2042,-49.7958,9E+09,9E+09,9E+09]];
     PERS ROBTARGET  SP_HCam_Side_YE := [[102.126,13.5,833.7],[6.88078E-09,0.956321,0.292317,-1.26749E-08],[-1,0,-1,0],[9E+09,-18.2042,-49.7958,9E+09,9E+09,9E+09]];
     PERS ROBTARGET  SP_HCam_Side_ZS := [[102.126,23.75,992.2],[0.676221,-0.676221,-0.206699,-0.206699],[0,-1,0,0],[9E+09,-18.2042,-49.7958,9E+09,9E+09,9E+09]];
     PERS ROBTARGET  SP_HCam_Side_ZE := [[102.126,23.75,942.2],[0.676221,-0.676221,-0.206699,-0.206699],[0,-1,0,0],[9E+09,-18.2042,-49.7958,9E+09,9E+09,9E+09]];
    !!!!!!!!!!!!!!!!!!!!!!!!!!!!!!!!!!!!!!!!!!
     PERS ROBTARGET  SP_GCam_Side_XS := [[-170.8,-16.55,-269.25],[0.328688,-0.328688,-0.62607,-0.62607],[-1,0,-3,0],[9E+09,-18.2042,49.7958,9E+09,9E+09,9E+09]];
     PERS ROBTARGET  SP_GCam_Side_XE := [[-120.8,-16.55,-269.25],[0.328688,-0.328688,-0.62607,-0.62607],[-1,0,-3,0],[9E+09,-18.2042,49.7958,9E+09,9E+09,9E+09]];
     PERS ROBTARGET  SP_GCam_Side_YS := [[-100.269,63.5,833.7],[9.15159E-09,0.648421,-0.761282,-3.15802E-08],[-1,0,-1,0],[9E+09,-18.2042,49.7958,9E+09,9E+09,9E+09]];
     PERS ROBTARGET  SP_GCam_Side_YE := [[-100.269,13.5,833.7],[9.15159E-09,0.648421,-0.761282,-3.15802E-08],[-1,0,-1,0],[9E+09,-18.2042,49.7958,9E+09,9E+09,9E+09]];
     PERS ROBTARGET  SP_GCam_Side_ZS := [[-100.269,23.75,992.2],[0.209515,-0.209515,0.675354,0.675354],[-1,0,0,1],[9E+09,-18.2042,49.7958,9E+09,9E+09,9E+09]];
     PERS ROBTARGET  SP_GCam_Side_ZE := [[-100.269,23.75,942.2],[0.209515,-0.209515,0.675354,0.675354],[-1,0,0,1],[9E+09,-18.2042,49.7958,9E+09,9E+09,9E+09]];
!!!!!!!!!!!!!!!!!!!!!!!!!!!!!!!!!!!!!!!!!!!!!!!!!!!!!!!!

    PERS robtarget SP_Hrnd_PJEDGE_S:=[[116.848,-37.6878,-156.792],[0.650768,-0.429986,0.562653,-0.273925],[-1,1,2,0],[9E+09,5.00003,90.0001,9E+09,9E+09,9E+09]];
	PERS robtarget SP_Hrnd_PJEDGE_E:=[[116.848,-37.6878,-131.792],[0.650768,-0.429986,0.562653,-0.273925],[-1,1,2,0],[9E+09,5.00003,90.0001,9E+09,9E+09,9E+09]];
    PERS robtarget SP_Hrnd_PjJOINT_S:=[[116.848,-37.1527,-150.737],[0.650775,-0.430009,0.56263,-0.273918],[-1,1,2,0],[9E+09,4.99996,89.9999,9E+09,9E+09,9E+09]];
    PERS robtarget SP_Hrnd_PjJOINT_E:=[[116.848,-37.1527,-125.737],[0.650775,-0.430009,0.56263,-0.273918],[-1,1,2,0],[9E+09,4.99996,89.9999,9E+09,9E+09,9E+09]];

    PERS robtarget SP_Grnd_PJEDGE_S:=[[-116.221,-37.9047,-158.274],[0.652633,0.0736842,-0.703268,-0.272131],[-1,-2,0,1],[9E+09,4.99994,-90.0001,9E+09,9E+09,9E+09]];
	PERS robtarget SP_Grnd_PJEDGE_E:=[[-116.221,-37.9047,-133.274],[0.652633,0.0736842,-0.703268,-0.272131],[-1,-2,0,1],[9E+09,4.99994,-90.0001,9E+09,9E+09,9E+09]];
    PERS robtarget SP_Grnd_PjJOINT_S:=[[-116.221,-37.2611,-151.785],[0.652662,0.0737409,-0.703265,-0.272052],[-1,-2,0,1],[9E+09,5.00007,-90.0001,9E+09,9E+09,9E+09]];
    PERS robtarget SP_Grnd_PjJOINT_E:=[[-116.221,-37.2611,-126.785],[0.652662,0.0737409,-0.703265,-0.272052],[-1,-2,0,1],[9E+09,5.00007,-90.0001,9E+09,9E+09,9E+09]];
    !!!!!!!!!!!!!!!!!!!!!!!!!!!!!!!!!!!!!!!!!!!!!!!!!!!!!!!!!!!!!!!!!!!!!

    PERS robtarget SP_GCAM_PJEDGE_S:=[[-105.775,-35.5,-136],[0.582944,-0.40023,0.582937,-0.400221],[-1,1,-2,0],[9E+09,0,90,9E+09,9E+09,9E+09]];
	PERS robtarget SP_GCAM_PJEDGE_E:=[[-105.775,-35.5,-106],[0.582969,-0.400229,0.582926,-0.400201],[-1,1,-2,0],[9E+09,0,89.9999,9E+09,9E+09,9E+09]];
    PERS robtarget SP_GCAM_PjJOINT_S:=[[-105.775,-35.5,-132],[0.670305,-0.384193,0.476249,-0.419849],[-1,1,-3,0],[9E+09,0,90,9E+09,9E+09,9E+09]];
    PERS robtarget SP_GCAM_PjJOINT_E:=[[-105.775,-35.5,-102],[0.670299,-0.384189,0.476254,-0.419857],[-1,1,-3,0],[9E+09,0,90,9E+09,9E+09,9E+09]];

    PERS robtarget SP_HCAM_PJEDGE_S:=[[108.602,-35.5,-136],[0.322637,-0.629197,-0.322659,0.629212],[-1,-4,3,1],[9E+09,0,-90,9E+09,9E+09,9E+09]];
	PERS robtarget SP_HCAM_PJEDGE_E:=[[108.602,-35.5,-106],[0.322651,-0.629208,-0.322631,0.629209],[-1,-4,3,1],[9E+09,0,-90,9E+09,9E+09,9E+09]];
    PERS robtarget SP_HCAM_PjJOINT_S:=[[108.602,-35.5,-132],[0.37527,-0.516211,-0.277231,0.718221],[-1,-4,3,1],[9E+09,0,-89.9999,9E+09,9E+09,9E+09]];
    PERS robtarget SP_HCAM_PjJOINT_E:=[[108.602,-35.5,-102],[0.375268,-0.516202,-0.277239,0.718225],[-1,-4,3,1],[9E+09,0,-90,9E+09,9E+09,9E+09]];
 !!
    PERS robtarget SP_PIV180_JOINT_E:=[[-0.0992797,10.0536,-155.969],[0.000391588,3.67936E-05,0.707076,-0.707138],[-1,1,-2,0],[9E+09,24.0001,180,9E+09,9E+09,9E+09]];
    PERS robtarget SP_PIV180_JOINT_S:=[[-0.0992797,10.0536,-180.969],[0.000391588,3.67936E-05,0.707076,-0.707138],[-1,1,-2,0],[9E+09,24.0001,180,9E+09,9E+09,9E+09]];
    PERS robtarget SP_PIV180_EDGE_E:=[[-0.357227,9.8351,-157.926],[0.000272799,0.000258098,0.707135,-0.707079],[-1,1,-2,0],[9E+09,24,180,9E+09,9E+09,9E+09]];
    PERS robtarget SP_PIV180_EDGE_S:=[[-0.357227,9.8351,-177.926],[0.000272799,0.000258098,0.707135,-0.707079],[-1,1,-2,0],[9E+09,24,180,9E+09,9E+09,9E+09]];

 !!!!!!!!!!!!!!!!!!!!!!!!!!!!!!!!!!!!!!!!!!!!!!!!!!!!!!!!!!!!!!!!!!!!!!!!!!!!!!!!!!!!!!!!!!!!!!!!!!!!!!!!

    PERS pose SRG_PJ_JOINT:=[[0,0.0154266,2.55237],[1,0,0,0]];
    PERS pose SRG_PJ_EDGE:=[[0,0.0548973,-0.643547],[1,0,0,0]];
    PERS pose SR_PIV180_EDGE:=[[0.669235,0,-0.248367],[1,0,0,0]];
    PERS pose SR_PIV180_JOINT:=[[0.669235,0,-0.440994],[1,0,0,0]];
    PERS pose SR_PIV180_X:=[[0,0,0],[1,0,0,0]];

  !!!!!!!!!!!!!!!!!!!!!!!!!!!!!!!!!!!!!!!!!!!!!!!!!!!!!!!!!!!!!!!!!!!!!!!!!!!!!!!!!!!!!!!!!!!!!!!!!!!!!!!
    PERS pose SRH_PJ_JOINT:=[[0,0.0363617,2.92647],[1,0,0,0]];
    PERS pose SRH_PJ_EDGE:=[[0,0.0869141,-0.68013],[1,0,0,0]];
!!!!!!@@@@@@@@@@@@@@@@@@@@@@@@@@@@@@@@@@@@@@@@@@@@@@@@@@@@@@@@@@@@@@@@@@@@@@@@@@@@@@@@@@@@@@@@@@@@@@@@@@@@@@@@@@@
!!!!!!@##########################################################################################################
!!!!!!... this is for an 18H part...!!!!!
!!!!!!...08-27-18 searches pointing towards tip!!!!!!!

!!!!!!!!!!!!!FOR 18H SEARCHES POINTING TOWARDS THE TIP (short wotox)
!!!!!!!!!!!!! TARGETS FOR THE ANCHORS!!!!!!!!!!!
!!!!!!!!!THESE robtargets reside IN EACH ACTUAL PART NUMBER MODULE!!!!!!!!!!!
	PERS robtarget SP_AGBY_S:=[[-37.2083,-53.5,-50],[0.866025,4.78467E-08,5.58349E-09,-0.5],[-1,-1,-1,0],[9E+09,0,-45,9E+09,9E+09,9E+09]];
	PERS robtarget SP_GX_S:=[[-52.7083,0,25],[0.683011,-0.683009,-0.183024,-0.183021],[-1,0,-1,0],[9E+09,0,-45,9E+09,9E+09,9E+09]];
	PERS robtarget SP_AGBZ_S:=[[-37.9583,60,43.5],[0.612382,-0.612379,-0.35354,-0.353538],[-1,0,-1,0],[9E+09,0,-45,9E+09,9E+09,9E+09]];
	PERS robtarget SP_AGFY_S:=[[-65,53.5,-170],[4.50996E-07,-0.707129,-0.707085,-4.27632E-08],[-1,-3,-1,0],[9E+09,-3.6377E-06,225,9E+09,9E+09,9E+09]];
	PERS robtarget SP_AGFZ_S:=[[-37.9583,-65,43.5],[0.533539,0.533559,0.464041,-0.464023],[0,-1,1,0],[9E+09,0,225,9E+09,9E+09,9E+09]];
	PERS robtarget SPAG205S:=[[-326.50,-11.52,205.07],[0.0462054,0.70654,0.0484451,0.704501],[0,0,-2,0],[9E+09,-2.85714E-05,90,9E+09,9E+09,9E+09]];

	PERS robtarget SP_AGBY_E:=[[-37.2083,-13.5,-50],[0.866025,4.78467E-08,5.58349E-09,-0.5],[-1,-1,-1,0],[9E+09,0,-45,9E+09,9E+09,9E+09]];
	PERS robtarget SP_GX_E:=[[-82.7083,0,25],[0.683011,-0.683009,-0.183024,-0.183021],[-1,0,-1,0],[9E+09,0,-45,9E+09,9E+09,9E+09]];
	PERS robtarget SP_AGBZ_E:=[[-37.9583,60,13.5],[0.612382,-0.612379,-0.35354,-0.353538],[-1,0,-1,0],[9E+09,0,-45,9E+09,9E+09,9E+09]];
	PERS robtarget SP_AGFY_E:=[[-65,13.5,-170],[4.50996E-07,-0.707129,-0.707085,-4.27632E-08],[-1,-3,-1,0],[9E+09,-3.6377E-06,225,9E+09,9E+09,9E+09]];
	PERS robtarget SP_AGFZ_E:=[[-37.9583,-65,13.5],[0.533539,0.533559,0.464041,-0.464023],[0,-1,1,0],[9E+09,0,225,9E+09,9E+09,9E+09]];
	PERS robtarget SPAG205E:=[[-326.50,-11.52,205.07],[0.0462054,0.70654,0.0484451,0.704501],[0,0,-2,0],[9E+09,-2.85714E-05,90,9E+09,9E+09,9E+09]];

	PERS robtarget SP_AHBY_S:=[[39.1189,-53.5,-50],[0.707169,1.61338E-06,-1.40706E-06,-0.707045],[-1,-2,0,0],[9E+09,0,45,9E+09,9E+09,9E+09]];
	PERS robtarget SP_HX_S:=[[54.6189,0,25],[0.435629,-0.435627,-0.556983,-0.55698],[-1,0,-2,0],[9E+09,0,45,9E+09,9E+09,9E+09]];
	PERS robtarget SP_AHBZ_S:=[[39.8689,60,43.5],[0.49741,-0.49744,-0.502577,-0.502547],[-1,0,-2,0],[9E+09,0,45,9E+09,9E+09,9E+09]];
	PERS robtarget SP_AHFY_S:=[[65,53.5,-170],[5.84915E-07,-0.707129,-0.707085,2.93282E-07],[-1,-4,0,0],[9E+09,-3.6377E-06,135,9E+09,9E+09,9E+09]];
	PERS robtarget SP_AHFZ_S:=[[39.8689,-65,43.5],[0.453292,0.45331,0.542706,-0.542686],[0,-1,1,0],[9E+09,0,135,9E+09,9E+09,9E+09]];
	PERS robtarget SPAH205S:=[[-326.50,-11.52,205.07],[0.0462054,0.70654,0.0484451,0.704501],[0,0,-2,0],[9E+09,-2.85714E-05,90,9E+09,9E+09,9E+09]];

	PERS robtarget SP_AHBY_E:=[[39.1189,-13.5,-50],[0.707169,1.61338E-06,-1.40706E-06,-0.707045],[-1,-2,0,0],[9E+09,0,45,9E+09,9E+09,9E+09]];
	PERS robtarget SP_HX_E:=[[84.6189,0,25],[0.435628,-0.435629,-0.556981,-0.556981],[-1,0,-2,0],[9E+09,0,45,9E+09,9E+09,9E+09]];
	PERS robtarget SP_AHBZ_E:=[[39.8689,60,13.5],[0.49741,-0.49744,-0.502577,-0.502547],[-1,0,-2,0],[9E+09,0,45,9E+09,9E+09,9E+09]];
	PERS robtarget SP_AHFY_E:=[[65,13.5,-170],[5.84915E-07,-0.707129,-0.707085,2.93282E-07],[-1,-4,0,0],[9E+09,-3.6377E-06,135,9E+09,9E+09,9E+09]];
	PERS robtarget SP_AHFZ_E:=[[39.8689,-65,13.5],[0.453292,0.45331,0.542706,-0.542686],[0,-1,1,0],[9E+09,0,135,9E+09,9E+09,9E+09]];
	PERS robtarget SPAH205E:=[[-326.50,-11.52,205.07],[0.0462054,0.70654,0.0484451,0.704501],[0,0,-2,0],[9E+09,-2.85714E-05,90,9E+09,9E+09,9E+09]];

!!!!!!!!!!!!!!!!!!!!NEW 03-25-18!!!!!!!!!!!!!!!!!!!!!!!!!!!!!!!!!!!!!!!!!!!!
!!!!!!!!!!!!!!!!!!!!!!!!!!!!!!!!!!!!!!!!! G & H ANCHOR FRONT X SEARCHES ! ADDED 3/25/18
	PERS robtarget SP_AGFX_E:=[[-82.7083,-50,43.5],[0.533539,0.533559,0.464041,-0.464023],[0,-1,1,0],[9E+09,0,225,9E+09,9E+09,9E+09]];
	PERS robtarget SP_AGFX_S:=[[-42.7083,-50,43.5],[0.533539,0.533559,0.464041,-0.464023],[0,-1,1,0],[9E+09,0,225,9E+09,9E+09,9E+09]];
	PERS robtarget AG_FX:=[[-43.5,-75,43.5],[0.533539,0.533559,0.464041,-0.464023],[0,-1,1,0],[9E+09,0,225,9E+09,9E+09,9E+09]];

    PERS robtarget SP_AHFX_S:=[[44.6189,-50,43.5],[0.453292,0.45331,0.542706,-0.542686],[0,-1,1,0],[9E+09,0,135,9E+09,9E+09,9E+09]];
	PERS robtarget SP_AHFX_E:=[[84.6189,-50,43.5],[0.453292,0.45331,0.542706,-0.542686],[0,-1,1,0],[9E+09,0,135,9E+09,9E+09,9E+09]];
	PERS robtarget AH_FX:=[[43.5,-75,13.5],[0.453292,0.45331,0.542706,-0.542686],[0,-1,1,0],[9E+09,0,135,9E+09,9E+09,9E+09]];

    PERS pose SR_AGF_X:=[[1.60019,-0.00982285,0.0090332],[1,0,0,0]];
    PERS pose SR_AHF_X:=[[-1.36459,0.000862122,0.00711441],[1,0,0,0]];

!!!!!!!!!!!!!!!!!!!!!!!!!!!!!!!!!!!!!!!!!!!!!!!!!!!!!!!!!!!!!!!!!!!!!!!!!!!!!!!!!!!!!!!


!!!!!!!!!!!!!!!!!!!  200'S ARE FOR SQUARE ANCHORS   !!!!!!!!!!!!!!!!!!!!!!!!!!!!!!!!!!
    PERS robtarget AG200:=[[-92.6081,-1.12,-59.77],[0.530075,-0.28296,-0.755868,-0.260032],[-1,0,-2,0],[9E+09,2.00003,-46.9999,9E+09,9E+09,9E+09]];
	PERS robtarget AG201:=[[-92.6081,-0.84,-67.99],[0.616379,-0.257434,-0.683208,-0.295013],[-1,0,-2,0],[9E+09,2,-46.9999,9E+09,9E+09,9E+09]];
	PERS robtarget AG202:=[[-92.6081,-2,-124],[0.670512,-0.228966,-0.634006,-0.309876],[-1,0,-2,0],[9E+09,2,-47,9E+09,9E+09,9E+09]];
	PERS robtarget AG203:=[[-92.6081,-0.93,-128.77],[0.705013,-0.0678415,-0.445609,0.547528],[0,1,-3,0],[9E+09,35,252,9E+09,9E+09,9E+09]];
	PERS robtarget AG204:=[[-92.6081,-17.55,-128.42],[0.707581,-0.0563974,-0.436894,0.552514],[0,1,-3,0],[9E+09,35,262,9E+09,9E+09,9E+09]];
	PERS robtarget AG205:=[[-92.6081,-31.58,-127.32],[0.695675,-0.0181838,-0.438224,0.568917],[0,1,-3,0],[9E+09,35,272,9E+09,9E+09,9E+09]];
	PERS robtarget AG206:=[[-92.6081,2,-64],[0.347708,-0.0611829,-0.822369,0.446166],[-1,1,-2,0],[9E+09,-2,227,9E+09,9E+09,9E+09]];
	PERS robtarget AG207:=[[-92.6081,3.62,-68],[0.414218,-0.0649739,-0.738676,0.527788],[-1,1,-2,0],[9E+09,-2,227,9E+09,9E+09,9E+09]];
	PERS robtarget AG208:=[[-92.6081,4.62,-124],[0.440384,-0.0595063,-0.689183,0.572318],[-1,1,-2,0],[9E+09,-1.99999,227,9E+09,9E+09,9E+09]];
	PERS robtarget AG209:=[[-92.6081,5.32575,-128.971],[0.443577,-0.0842176,-0.714974,0.533816],[-1,1,-2,0],[9E+09,-0.65,-133.55,9E+09,9E+09,9E+09]];
    PERS robtarget AG210:=[[-92.6081,-13.5816,-138.756],[0.641565,0.44099,0.276145,0.563619],[0,0,-3,0],[9E+09,39.5072,-243.585,9E+09,9E+09,9E+09]];
	PERS robtarget AG218:=[[-92.6081,-30.49,-54.53],[0.0709792,0.698666,0.59999,-0.383197],[0,2,-2,0],[9E+09,-35,278,9E+09,9E+09,9E+09]];
	PERS robtarget AG219:=[[-92.6081,-16.69,-55.74],[0.0149731,0.717884,0.581263,-0.382821],[0,2,-2,0],[9E+09,-35,268,9E+09,9E+09,9E+09]];
    PERS robtarget AG220:=[[-92.6081,0.86,-58.5],[0.0438935,-0.740378,-0.559595,0.36982],[0,2,-2,0],[9E+09,-35,258,9E+09,9E+09,9E+09]];

	PERS robtarget AH200:=[[94.7543,-1.63,-60.67],[0.426143,-0.801361,-0.0154398,-0.419504],[-1,1,-2,0],[9E+09,2.00003,46.9999,9E+09,9E+09,9E+09]];
	PERS robtarget AH201:=[[94.7543,-2,-68],[0.508529,-0.721626,-0.03114,-0.468704],[-1,1,-2,0],[9E+09,2,47,9E+09,9E+09,9E+09]];
	PERS robtarget AH202:=[[94.7543,-2,-124],[0.54208,-0.669718,-0.0329965,-0.506497],[-1,1,-2,0],[9E+09,2,47,9E+09,9E+09,9E+09]];
	PERS robtarget AH203:=[[94.7543,-2.04,-127.84],[0.404162,0.415064,-0.0538961,0.813308],[-1,0,-2,0],[9E+09,35,105,9E+09,9E+09,9E+09]];
	PERS robtarget AH204:=[[94.7543,-21.37,-127.81],[0.419692,0.403161,-0.0745871,0.809788],[-1,0,-2,0],[9E+09,35,95,9E+09,9E+09,9E+09]];
	PERS robtarget AH205:=[[94.7543,-31.34,-128.11],[0.433629,0.405743,-0.112626,0.796651],[0,0,-2,0],[9E+09,35,79.9999,9E+09,9E+09,9E+09]];
	PERS robtarget AH206:=[[94.7543,2,-64],[0.473198,0.788653,0.294146,0.259978],[-1,0,-3,0],[9E+09,-2,137,9E+09,9E+09,9E+09]];
	PERS robtarget AH207:=[[94.7543,3.59,-67.98],[0.614532,0.681338,0.316142,0.241211],[0,0,-3,0],[9E+09,-1.99998,137,9E+09,9E+09,9E+09]];
	PERS robtarget AH208:=[[94.7543,3.15,-123.6],[0.692906,0.609033,0.263193,0.282292],[0,0,-2,0],[9E+09,-2.00002,137,9E+09,9E+09,9E+09]];
	PERS robtarget AH209:=[[94.7543,5.32575,-128.971],[0.559127,0.667651,0.114895,0.477933],[-1,0,-2,0],[9E+09,8.22046,-231.454,9E+09,9E+09,9E+09]];
    PERS robtarget AH210:=[[94.7543,-13.5816,-138.756],[0.568028,0.631405,0.131371,0.511288],[0,0,-2,0],[9E+09,88.8261,-234.061,9E+09,9E+09,9E+09]];
	PERS robtarget AH218:=[[94.7543,-32.41,-55.09],[0.345707,0.311744,0.848036,-0.253255],[0,-1,-3,0],[9E+09,-35,86.9999,9E+09,9E+09,9E+09]];
	PERS robtarget AH219:=[[94.7543,-15.87,-55.29],[0.373932,0.279544,0.863907,-0.188928],[0,-1,-3,0],[9E+09,-35,97,9E+09,9E+09,9E+09]];
    PERS robtarget AH220:=[[94.7543,-4.5,-56.5],[0.427902,0.243855,0.857844,-0.146764],[0,-1,-3,0],[9E+09,-35,107,9E+09,9E+09,9E+09]];


    !!!!!!!!!!!!!!300'S ARE FOR AN H ANCHOR!!!!!!!!!!!!!!!!!!!!!!!!!!!!!!!!!!!!!!!!!!!!!!!!!!!!!!!!!!!!!!!!!!!!!!!!!!!!!!!!!!!!!!!!
    PERS robtarget AH300:=[[94.7543,-6.57,-21.73],[0.41253,-0.781267,0.0558309,-0.465106],[-1,1,-2,0],[9E+09,8.00001,40.6874,9E+09,9E+09,9E+09]];
    PERS robtarget AH301:=[[94.7543,-6.58,-28.82],[0.471057,-0.721347,0.0463554,-0.505584],[-1,1,-2,0],[9E+09,8.00001,40.6874,9E+09,9E+09,9E+09]];
    PERS robtarget AH302:=[[94.7543,-5.48,-91.96],[0.471062,-0.72135,0.046355,-0.505575],[0,1,-2,0],[9E+09,8.00001,40.6871,9E+09,9E+09,9E+09]];
    PERS robtarget AH303:=[[94.7543,-0.85,-110.45],[0.520826,-0.563523,0.137798,-0.626253],[0,2,-3,0],[9E+09,2.59754E-05,91.7027,9E+09,9E+09,9E+09]];
    PERS robtarget AH304:=[[94.7543,13.67,-116.63],[0.528651,-0.508877,0.129899,-0.666857],[0,2,-3,0],[9E+09,-2.5987E-05,89.6851,9E+09,9E+09,9E+09]];
    PERS robtarget AG300:=[[-92.6081,-10.14,-20.37],[0.59256,-0.251762,-0.724769,-0.245355],[-1,0,-2,0],[9E+09,8.00001,-40.6872,9E+09,9E+09,9E+09]];
    PERS robtarget AG301:=[[-92.6081,-6.37,-25.55],[0.62849,-0.208495,-0.715362,-0.223132],[-1,0,-2,0],[9E+09,7.99998,-40.6871,9E+09,9E+09,9E+09]];
    PERS robtarget AG303:=[[-92.6081,-2.05,-109.81],[0.778403,-0.146079,-0.568319,-0.223077],[0,0,-2,0],[9E+09,-2.5987E-05,-70.2826,9E+09,9E+09,9E+09]];
    PERS robtarget AG304:=[[-92.6081,12.41,-117.42],[0.861143,-0.0506797,-0.481908,-0.153721],[0,0,-2,0],[9E+09,2.59754E-05,-95.5651,9E+09,9E+09,9E+09]];
    PERS robtarget AG302:=[[-92.6081,-6.38,-97.25],[0.628487,-0.208491,-0.715365,-0.223134],[-1,0,-2,0],[9E+09,8.00001,-40.6872,9E+09,9E+09,9E+09]];
    PERS robtarget AG306:=[[-92.6081,3.97,-17.51],[0.393636,-0.0526268,-0.758786,0.51626],[-1,1,-2,0],[9E+09,-3,220.687,9E+09,9E+09,9E+09]];
    PERS robtarget AG307:=[[-92.6081,4.38,-21.71],[0.447231,-0.0785861,-0.701275,0.549565],[-1,1,-2,0],[9E+09,-3,220.687,9E+09,9E+09,9E+09]];
    PERS robtarget AG308:=[[-92.6081,4.4,-90.43],[0.447233,-0.0785877,-0.701276,0.549562],[0,1,-2,0],[9E+09,-3,220.687,9E+09,9E+09,9E+09]];
    PERS robtarget AG309:=[[-92.6081,1.28,-107.03],[0.569535,-0.0958386,-0.560521,0.593517],[0,1,-3,0],[9E+09,2.59754E-05,243.45,9E+09,9E+09,9E+09]];
    PERS robtarget AG310:=[[-92.6081,-10.69,-114.74],[0.625255,-0.132271,-0.50974,0.575957],[0,2,-3,0],[9E+09,-5.20202E-06,261.9,9E+09,9E+09,9E+09]];
    PERS robtarget AH306:=[[94.7543,4.84,-16.92],[0.393381,0.795722,0.095828,0.450439],[-1,0,-3,0],[9E+09,-3,139.313,9E+09,9E+09,9E+09]];
    PERS robtarget AH307:=[[94.7543,4.85,-20.44],[0.483214,0.739516,0.0447349,0.466497],[-1,0,-2,0],[9E+09,-3,139.313,9E+09,9E+09,9E+09]];
    PERS robtarget AH308:=[[94.7543,4.86,-91.47],[0.483212,0.739515,0.0447391,0.466499],[-1,0,-2,0],[9E+09,-3,139.313,9E+09,9E+09,9E+09]];
    PERS robtarget AH309:=[[94.7543,0.88,-105.94],[0.390951,0.641757,-0.0550254,0.657478],[-1,0,-2,0],[9E+09,-1.49997,116.682,9E+09,9E+09,9E+09]];
    PERS robtarget AH310:=[[94.7543,-11.18,-111.14],[0.224534,0.514984,-0.062495,0.824906],[0,0,-2,0],[9E+09,-5.20202E-06,94.05,9E+09,9E+09,9E+09]];

 !!!!!!!!!!!!!!!!!!!  400'S ARE FOR 100F SQUARE ANCHORS with TAPERED EARS AND WOBJS  !!!!!!!!!!!!!!!!!!!!!!!!!!!!!!!!!!
    PERS robtarget AG400:=[[-92.6081,13.73,-90.65],[0.548124,-0.271296,-0.748356,-0.256754],[-1,0,-2,0],[9E+09,-0.899984,-44.0513,9E+09,9E+09,9E+09]];
	PERS robtarget AG401:=[[-92.6081,13.95,-95.56],[0.594775,-0.265788,-0.702359,-0.286865],[-1,0,-2,0],[9E+09,-0.899984,-44.0513,9E+09,9E+09,9E+09]];
	PERS robtarget AG402:=[[-92.6081,7.55,-179.34],[0.639524,-0.241649,-0.667142,-0.295867],[-1,0,-2,0],[9E+09,-0.900004,-44.0513,9E+09,9E+09,9E+09]];
	PERS robtarget AG403:=[[-92.6081,11.61,-176.06],[0.712014,-0.112487,-0.434654,0.539869],[-1,1,-3,0],[9E+09,35,270.049,9E+09,9E+09,9E+09]];
	PERS robtarget AG404:=[[-92.6081,-13.5,-183],[0.725082,-0.12027,-0.402489,0.545705],[-1,1,-3,0],[9E+09,35,270.049,9E+09,9E+09,9E+09]];
	PERS robtarget AG405:=[[-92.6081,-37.52,-188.39],[0.718927,-0.0817298,-0.401172,0.561716],[-1,1,-3,0],[9E+09,35,270.049,9E+09,9E+09,9E+09]];
	PERS robtarget AG406:=[[-92.6081,-15.92,-81.78],[0.357787,-0.0905625,-0.817756,0.441659],[-1,1,-2,0],[9E+09,-0.0487044,225.949,9E+09,9E+09,9E+09]];
	PERS robtarget AG407:=[[-92.6081,-13.49,-92.11],[0.402308,-0.0725723,-0.752787,0.515939],[-1,1,-2,0],[9E+09,-0.0487044,225.949,9E+09,9E+09,9E+09]];
	PERS robtarget AG408:=[[-92.6081,6.62,-169.15],[0.408311,-0.0639001,-0.735888,0.536346],[-1,1,-2,0],[9E+09,-0.0486628,225.949,9E+09,9E+09,9E+09]];
	PERS robtarget AG409:=[[-92.6081,5.32575,-128.971],[0.443577,-0.0842176,-0.714974,0.533816],[-1,1,-2,0],[9E+09,-0.65,-133.55,9E+09,9E+09,9E+09]];
    PERS robtarget AG410:=[[-92.6081,-13.5816,-138.756],[0.641565,0.44099,0.276145,0.563619],[0,0,-3,0],[9E+09,39.5072,-243.585,9E+09,9E+09,9E+09]];
	PERS robtarget AG418:=[[-92.6081,-65.74,-81.68],[0.19119,-0.713664,-0.622944,0.257042],[-1,1,-2,0],[9E+09,-35,269.951,9E+09,9E+09,9E+09]];
	PERS robtarget AG419:=[[-92.6081,-41.96,-76.74],[0.165424,-0.714306,-0.612118,0.296166],[-1,1,-2,0],[9E+09,-35,269.951,9E+09,9E+09,9E+09]];
    PERS robtarget AG420:=[[-92.6081,-18.08,-72.74],[0.192126,-0.708168,-0.606324,0.306524],[-1,1,-2,0],[9E+09,-35,269.951,9E+09,9E+09,9E+09]];

	PERS robtarget AH400:=[[94.7543,13.33,-93.75],[0.393162,-0.817804,0.00997615,-0.420144],[-1,1,-2,0],[9E+09,-0.900004,44.0512,9E+09,9E+09,9E+09]];
	PERS robtarget AH401:=[[94.7543,13.69,-101.41],[0.487688,-0.72347,-0.0068602,-0.488574],[-1,1,-2,0],[9E+09,-0.900004,44.0513,9E+09,9E+09,9E+09]];
	PERS robtarget AH402:=[[94.7543,9.58,-182.62],[0.496926,-0.708351,-0.00192019,-0.501298],[-1,1,-2,0],[9E+09,-0.900004,44.0514,9E+09,9E+09,9E+09]];
	PERS robtarget AH403:=[[94.7543,7.57,-176.59],[0.423025,0.451141,0.0368039,0.784963],[-1,0,-2,0],[9E+09,35,89.9513,9E+09,9E+09,9E+09]];
	PERS robtarget AH404:=[[94.7543,-15.09,-183.47],[0.430206,0.460496,0.0137373,0.776323],[-1,0,-2,0],[9E+09,35,89.9513,9E+09,9E+09,9E+09]];
	PERS robtarget AH405:=[[94.7543,-33.73,-187.06],[0.435284,0.430806,0.0148724,0.790388],[-1,0,-2,0],[9E+09,35,89.9513,9E+09,9E+09,9E+09]];
	PERS robtarget AH406:=[[94.7543,-17.23,-85.51],[0.475286,0.786592,0.287429,0.269742],[-1,0,-3,0],[9E+09,-0.0487252,134.051,9E+09,9E+09,9E+09]];
	PERS robtarget AH407:=[[94.7543,-13.59,-94.34],[0.57934,0.699674,0.34533,0.235729],[-1,-1,-3,0],[9E+09,-0.0486836,134.051,9E+09,9E+09,9E+09]];
	PERS robtarget AH408:=[[94.7543,3.51,-174.37],[0.649884,0.646412,0.309789,0.252651],[-1,-1,-2,0],[9E+09,-0.0487044,134.051,9E+09,9E+09,9E+09]];
	PERS robtarget AH409:=[[94.7543,5.32575,-128.971],[0.559127,0.667651,0.114895,0.477933],[-1,0,-2,0],[9E+09,8.22046,-231.454,9E+09,9E+09,9E+09]];
    PERS robtarget AH410:=[[94.7543,-13.5816,-138.756],[0.568028,0.631405,0.131371,0.511288],[0,0,-2,0],[9E+09,88.8261,-234.061,9E+09,9E+09,9E+09]];
	PERS robtarget AH418:=[[94.7543,-65.46,-88.56],[0.268952,0.667819,0.674236,0.164586],[-1,-1,-3,0],[9E+09,-35,90.0488,9E+09,9E+09,9E+09]];
	PERS robtarget AH419:=[[94.7543,-37.27,-83.18],[0.276819,0.653558,0.674141,0.204369],[-1,-1,-3,0],[9E+09,-35,90.0487,9E+09,9E+09,9E+09]];
    PERS robtarget AH420:=[[94.7543,-16.85,-79.86],[0.284029,0.647089,0.671745,0.222175],[-1,-1,-3,0],[9E+09,-35,90.0487,9E+09,9E+09,9E+09]];

    !!!!!!!!!!!!!!!!!!!  38H AND 42H ANCHORS with TAPERED EARS AND WOBJS  !!!!!!!!!!!!!!!!!!!!!!!!!!!!!!!!!!
    PERS robtarget AG500:=[[-119.5,-19.0771,7.8546],[0.18894,-0.393143,-0.665153,0.606062],[-1,2,2,0],[9E+09,-1,229.037,9E+09,9E+09,9E+09]];
	PERS robtarget AG501:=[[-119.5,-21.4179,18.2494],[0.177597,-0.397618,-0.681839,0.587754],[-1,2,2,0],[9E+09,-1,229.037,9E+09,9E+09,9E+09]];
	PERS robtarget AG502:=[[-119.5,-37.2938,40.053],[0.1671,-0.537437,-0.637802,0.525782],[-1,1,2,0],[9E+09,-20.9627,243.463,9E+09,9E+09,9E+09]];
	PERS robtarget AG503:=[[-119.5,-64.056,43.4312],[0.197414,-0.658472,-0.572464,0.446908],[-1,1,2,0],[9E+09,-20.9627,265.963,9E+09,9E+09,9E+09]];
	PERS robtarget AG504:=[[-119.5,-1.87894,-73.1379],[0.408467,-0.108421,-0.754714,0.501804],[-1,1,2,0],[9E+09,-1,229.037,9E+09,9E+09,9E+09]];
	PERS robtarget AG505:=[[-119.5,3.83214,-100.279],[0.412665,-0.111226,-0.752426,0.50119],[-1,1,2,0],[9E+09,-1,229.037,9E+09,9E+09,9E+09]];
	PERS robtarget AG506:=[[-119.5,-0.673835,-119.593],[0.470803,-0.169688,-0.576014,0.646342],[-1,2,1,0],[9E+09,20.9627,251.537,9E+09,9E+09,9E+09]];
	PERS robtarget AG507:=[[-119.5,-17.226,-130.381],[0.665958,-0.157931,-0.512595,0.518463],[-1,1,1,0],[9E+09,20.9627,274.037,9E+09,9E+09,9E+09]];
	PERS robtarget AG508:=[[-119.5,32.0542,48.9725],[0.170455,0.80062,-0.424285,-0.387213],[-1,1,-1,1],[9E+09,-20.9627,-94.0373,9E+09,9E+09,9E+09]];
	PERS robtarget AG509:=[[-119.5,6.68673,39.7911],[0.0933594,0.711654,-0.449901,-0.531434],[-1,1,-1,1],[9E+09,-20.9627,-63.4627,9E+09,9E+09,9E+09]];
    PERS robtarget AG510:=[[-119.5,-4,15.04],[0.0199359,-0.565142,0.460583,0.684163],[-1,1,-1,1],[9E+09,1,-40.9627,9E+09,9E+09,9E+09]];
    PERS robtarget AG511:=[[-119.5,-4,-52.5],[0.0133879,-0.53789,0.460896,0.705741],[-1,1,-1,1],[9E+09,1,-40.9627,9E+09,9E+09,9E+09]];
    PERS robtarget AG512:=[[-119.50,-4.00,-47.50],[0.662788,-0.305779,-0.658678,-0.182632],[-1,-2,0,1],[9E+09,1,-40.9627,9E+09,9E+09,9E+09]];
	PERS robtarget AG513:=[[-119.50,-4.00,-99.96],[0.651392,-0.315816,-0.664542,-0.185287],[-1,-2,0,1],[9E+09,1,-40.9627,9E+09,9E+09,9E+09]];
    PERS robtarget AG514:=[[-119.5,3.33891,-118.463],[0.788634,-0.133339,-0.551103,-0.237829],[-1,-2,0,1],[9E+09,20.9627,-63.4627,9E+09,9E+09,9E+09]];
    PERS robtarget AG515:=[[-119.5,21.3558,-126.913],[0.804002,-0.0544646,-0.498961,-0.31883],[-1,-2,0,1],[9E+09,20.9627,-85.9627,9E+09,9E+09,9E+09]];
	PERS robtarget AH500:=[[119.5,-19.0771,7.8546],[0.605344,0.645275,0.402981,0.234063],[-1,-1,1,0],[9E+09,-1,130.963,9E+09,9E+09,9E+09]];
	PERS robtarget AH501:=[[119.5,-21.4179,18.2494],[0.604403,0.656405,0.347311,0.288453],[-1,-1,1,0],[9E+09,-1,130.963,9E+09,9E+09,9E+09]];
	PERS robtarget AH502:=[[119.5,-37.2938,40.053],[0.359554,0.756138,0.484145,0.254127],[-1,-1,1,0],[9E+09,-20.9627,116.537,9E+09,9E+09,9E+09]];
	PERS robtarget AH503:=[[119.5,-64.056,43.4312],[0.307627,0.721493,0.575875,0.230609],[-1,-1,1,0],[9E+09,-20.9627,94.0373,9E+09,9E+09,9E+09]];
	PERS robtarget AH504:=[[119.5,-1.87894,-73.1379],[0.420104,0.747691,0.0630285,0.510391],[-1,0,2,0],[9E+09,-1,130.963,9E+09,9E+09,9E+09]];
	PERS robtarget AH505:=[[119.5,3.83214,-100.279],[0.420104,0.747691,0.0630288,0.51039],[-1,0,2,0],[9E+09,-1,130.963,9E+09,9E+09,9E+09]];
	PERS robtarget AH506:=[[119.5,-0.673835,-119.593],[0.429458,0.631672,0.006994,0.645374],[-1,0,2,0],[9E+09,10,108.463,9E+09,9E+09,9E+09]];
	PERS robtarget AH507:=[[119.5,-17.226,-130.381],[0.365774,0.502624,0.0139829,0.783188],[-1,0,2,0],[9E+09,20.9627,85.9627,9E+09,9E+09,9E+09]];
	PERS robtarget AH508:=[[119.5,32.0542,48.9725],[0.22927,-0.690268,0.587125,-0.355316],[-1,1,-2,0],[9E+09,-20.9627,84.0373,9E+09,9E+09,9E+09]];
	PERS robtarget AH509:=[[119.5,6.68673,39.7911],[0.466815,-0.683703,0.519973,-0.210387],[-1,1,-2,0],[9E+09,-20.9627,63.4627,9E+09,9E+09,9E+09]];
    PERS robtarget AH510:=[[119.5,-4,15.04],[0.6885,-0.592606,0.40062,-0.119534],[-1,2,-2,0],[9E+09,1,40.9627,9E+09,9E+09,9E+09]];
    PERS robtarget AH511:=[[119.5,-4,-52.5],[0.679627,-0.590707,0.425456,-0.090328],[-1,2,-2,0],[9E+09,1,40.9627,9E+09,9E+09,9E+09]];
    PERS robtarget AH512:=[[119.5,-4,-47.5],[0.532284,-0.698007,0.0487269,-0.476536],[-1,1,-2,0],[9E+09,1,40.9627,9E+09,9E+09,9E+09]];
	PERS robtarget AH513:=[[119.5,-4,-99.96],[0.554206,-0.665717,0.0487589,-0.497292],[-1,1,-2,0],[9E+09,1,40.9627,9E+09,9E+09,9E+09]];
    PERS robtarget AH514:=[[119.5,3.33891,-118.463],[0.488848,-0.5234,0.0681067,-0.694581],[-1,1,-3,0],[9E+09,20.9627,63.4627,9E+09,9E+09,9E+09]];
    PERS robtarget AH515:=[[119.5,21.3558,-126.913],[0.395971,-0.4509,0.0152689,-0.799789],[-1,1,-3,0],[9E+09,20.9627,85.9627,9E+09,9E+09,9E+09]];
!!!!!!!!!!!!!SEARCHSTOP'S FOR SNIFFING THE ANCHOR WORK OBJECT!!!!!!!!!!!!!!!!!!!!!


!!!!!!!!!!!!!!!!!!!!!!!!!!!!!!!!!!!!!!!!!!!!!!!!!!!!!ROBTARGETS!!!!!!!!!!!!!!!!!!!!!!!!!!!!!!!!!!!!!!!!!!!!!!!!!!!!!!!!!!!!!!!!!!!!!!
!!!!!!!!!!!!!!!!!!!!!!!!!!!!!!!!!!!!!!!!!!!!!!!!!!!!!ROBTARGETS!!!!!!!!!!!!!!!!!!!!!!!!!!!!!!!!!!!!!!!!!!!!!!!!!!!!!!!!!!!!!!!!!!!!!!
!!!!!!!!!!!!WRAPPER WELDS!!
!!!!!!!!!!!!!!!!!!!!!!!!!!!!!!!!!!!!!!!!!!!!!!!!!!!!!ROBTARGETS!!!!!!!!!!!!!!!!!!!!!!!!!!!!!!!!!!!!!!!!!!!!!!!!!!!!!!!!!!!!!!!!!!!!!!
	PERS robtarget A33K:=[[0,-380.805,718.334],[0.281446,-0.295038,-0.645509,0.645801],[-1,1,-2,0],[9E+09,0.275255,-133.775,9E+09,9E+09,9E+09]];
	PERS robtarget A36K:=[[0,-335.444,444.288],[0.328875,-0.233147,-0.765099,0.502102],[-1,1,-2,0],[9E+09,-15.5279,-130.528,9E+09,9E+09,9E+09]];
	PERS robtarget B33K:=[[0,-406.805,718.334],[0.310377,-0.311928,0.64637,-0.623356],[-1,1,-3,0],[9E+09,0.275255,133.775,9E+09,9E+09,9E+09]];
	PERS robtarget B36K:=[[0,-361.444,444.288],[0.344577,-0.25808,0.752135,-0.498954],[0,2,-2,0],[9E+09,-15.5279,130.528,9E+09,9E+09,9E+09]];
	PERS robtarget G15K:=[[0,-294.296,553.194],[0.667793,-0.60282,0.336004,-0.278857],[-1,2,-3,0],[9E+09,4.35425,47.6458,9E+09,9E+09,9E+09]];
	PERS robtarget G21K:=[[0,-300.481,733.133],[0.621746,-0.655911,0.304929,-0.300384],[-1,1,-2,0],[9E+09,-1.26795,46.7321,9E+09,9E+09,9E+09]];
	PERS robtarget H15K:=[[0,-284.696,553.194],[0.672577,-0.593354,-0.333612,0.290301],[-1,1,-2,0],[9E+09,4.35425,-47.6458,9E+09,9E+09,9E+09]];
	PERS robtarget H21K:=[[0,-290.881,733.133],[0.607609,-0.6571,-0.312229,0.318659],[-1,1,-2,0],[9E+09,-1.26795,-46.7321,9E+09,9E+09,9E+09]];
	PERS robtarget L64K:=[[97.4377,-290.285,611.781],[0.668128,-0.628289,0.296316,-0.266561],[-1,1,-2,0],[9E+09,2,47,9E+09,9E+09,9E+09]];
	PERS robtarget L65K:=[[97.0147,-281.034,526.913],[0.6909,-0.599747,0.302731,-0.267047],[-1,2,-3,0],[9E+09,5.58452,47.9155,9E+09,9E+09,9E+09]];
	PERS robtarget L66K:=[[96.6555,-267.246,454.85],[0.721323,-0.562078,0.320083,-0.247605],[0,2,-3,0],[9E+09,9.39445,48.6055,9E+09,9E+09,9E+09]];
	PERS robtarget L67K:=[[96.5969,-264.534,443.099],[0.723995,-0.558714,0.320175,-0.2473],[0,2,-3,0],[9E+09,9.82577,48.6742,9E+09,9E+09,9E+09]];
	PERS robtarget M64K:=[[-92.2808,-290.285,611.781],[0.643983,-0.197754,-0.665916,-0.320523],[-1,0,-2,0],[9E+09,2,-47,9E+09,9E+09,9E+09]];
	PERS robtarget M65K:=[[-92.0438,-281.034,526.913],[0.640466,-0.138859,-0.657313,-0.372102],[-1,0,-2,0],[9E+09,5.58452,-47.9155,9E+09,9E+09,9E+09]];
	PERS robtarget M66K:=[[-92.4965,-267.246,454.85],[0.659146,-0.125605,-0.634514,-0.38359],[-1,0,-2,0],[9E+09,9.39445,-48.6055,9E+09,9E+09,9E+09]];
	PERS robtarget M67K:=[[-92.5824,-264.534,443.099],[0.669311,-0.137751,-0.629046,-0.370607],[-1,0,-2,0],[9E+09,9.82577,-48.6742,9E+09,9E+09,9E+09]];





!!!!!!!!!!!!WRAPPER WELDS!!
	PERS robtarget A30:=[[0,-263.6,571.811],[0.301458,-0.366237,-0.576552,0.665268],[-1,2,-2,0],[9E+09,8.10886,-131.609,9E+09,9E+09,9E+09]];
	PERS robtarget A31:=[[0,-364.406,856.989],[0.251716,-0.313959,-0.586031,0.703303],[-1,1,-2,0],[9E+09,8.5359,-131.536,9E+09,9E+09,9E+09]];
	PERS robtarget A32:=[[0,-271.562,492.705],[0.338101,-0.313827,-0.640016,0.614475],[-1,1,-2,0],[9E+09,-0.207117,-134.293,9E+09,9E+09,9E+09]];
	PERS robtarget A325:=[[0,-157.742,344.172],[0.35801,-0.217133,-0.6963,0.582966],[0,1,-2,0],[9E+09,-22.95,-129.52,9E+09,9E+09,9E+09]];
	PERS robtarget A33:=[[0,-270.812,423.864],[0.364589,-0.288048,-0.679272,0.568061],[0,1,-2,0],[9E+09,-6.41778,-131.918,9E+09,9E+09,9E+09]];
	PERS robtarget A34:=[[0,-263.637,413.741],[0.366015,-0.285193,-0.700771,0.541865],[0,1,-2,0],[9E+09,-7.68339,-131.683,9E+09,9E+09,9E+09]];
	PERS robtarget A35:=[[0,-339.363,455.358],[0.344164,-0.221752,-0.741689,0.531295],[-1,1,-2,0],[9E+09,-14.6411,-130.641,9E+09,9E+09,9E+09]];
	PERS robtarget A36:=[[0,-245.168,337.254],[0.4087,-0.251395,-0.719948,0.501437],[0,1,-2,0],[9E+09,-11,-130.257,9E+09,9E+09,9E+09]];
	PERS robtarget A37:=[[0,-275.3,318.511],[0.346619,-0.1901,-0.797309,0.456087],[0,1,-2,0],[9E+09,-25.4322,-129.432,9E+09,9E+09,9E+09]];
	PERS robtarget A38:=[[0,-207.054,267.395],[0.419939,-0.214995,-0.766545,0.435704],[0,1,-2,0],[9E+09,-17,-129.169,9E+09,9E+09,9E+09]];
    PERS robtarget A39:=[[0,-175.384,220.232],[0.419924,-0.214999,-0.766549,0.435709],[0,1,-2,0],[9E+09,-17,-129.169,9E+09,9E+09,9E+09]];
    PERS robtarget A395:=[[107.03,-70.02,238.50],[0.373597,-0.290524,-0.671191,0.570546],[0,1,-2,0],[9E+09,-17,-129.195,9E+09,9E+09,9E+09]];
    PERS robtarget A395L:=[[111.42,-51.07,166.04],[0.355193,-0.283718,-0.689611,0.563718],[0,1,-2,0],[9E+09,-17,-129.195,9E+09,9E+09,9E+09]];
    PERS robtarget A395R:=[[113.65,-57.02,158.59],[0.355422,-0.28373,-0.659728,0.598275],[0,1,-2,0],[9E+09,-27.8948,-129.195,9E+09,9E+09,9E+09]];
    PERS robtarget A395S:=[[113.65,-57.02,158.6],[0.355419,-0.283731,-0.659728,0.598276],[0,1,-2,0],[9E+09,-27.8948,-129.195,9E+09,9E+09,9E+09]];

	PERS robtarget B30:=[[0,-267.178,571.9],[0.291352,-0.33181,0.574241,-0.689394],[-1,1,-3,0],[9E+09,8.10884,131.609,9E+09,9E+09,9E+09]];
	PERS robtarget B31:=[[0,-390.406,856.989],[0.277445,-0.357674,0.57458,-0.681874],[-1,1,-3,0],[9E+09,8.5359,131.536,9E+09,9E+09,9E+09]];
	PERS robtarget B32:=[[0,-274.839,492.688],[0.319301,-0.293352,0.64875,-0.625392],[0,2,-2,0],[9E+09,-0.207117,134.293,9E+09,9E+09,9E+09]];
	PERS robtarget B325:=[[0,-181.423,339.977],[0.317696,-0.339484,0.642994,-0.608588],[0,2,-2,0],[9E+09,-22.95,140.48,9E+09,9E+09,9E+09]];
	PERS robtarget B33:=[[0,-268.33,424.285],[0.351184,-0.26984,0.694036,-0.5676],[0,2,-2,0],[9E+09,-6.41779,131.918,9E+09,9E+09,9E+09]];
	PERS robtarget B34:=[[0,-266.897,413.708],[0.348878,-0.26926,0.711428,-0.547406],[0,2,-2,0],[9E+09,-7.68338,131.683,9E+09,9E+09,9E+09]];
	PERS robtarget B35:=[[0,-365.363,455.358],[0.355113,-0.246559,0.73281,-0.525445],[0,2,-2,0],[9E+09,-14.6411,130.641,9E+09,9E+09,9E+09]];
	PERS robtarget B36:=[[0,-243.624,337.924],[0.366083,-0.240661,0.738256,-0.512878],[0,2,-2,0],[9E+09,-11,130.257,9E+09,9E+09,9E+09]];
	PERS robtarget B37:=[[0,-301.3,318.511],[0.380085,-0.204643,0.782357,-0.448969],[0,2,-2,0],[9E+09,-25.4322,129.432,9E+09,9E+09,9E+09]];
	PERS robtarget B38:=[[0,-206.544,267.658],[0.410849,-0.214317,0.775145,-0.429443],[0,2,-2,0],[9E+09,-17.0001,129.169,9E+09,9E+09,9E+09]];
    PERS robtarget B39:=[[0,-174.984,220.467],[0.391153,-0.203413,0.785267,-0.434716],[0,2,-2,0],[9E+09,-17,129.169,9E+09,9E+09,9E+09]];
    PERS robtarget B395:=[[-112.59,-71.04,233.12],[0.368967,-0.296309,0.682077,-0.557526],[0,2,-2,0],[9E+09,-17,129.195,9E+09,9E+09,9E+09]];
    PERS robtarget B395L:=[[-114.28,-54.25,162.26],[0.373526,-0.287657,0.69003,-0.549172],[0,2,-2,0],[9E+09,-17,129.195,9E+09,9E+09,9E+09]];
    PERS robtarget B395R:=[[-109.29,-57.86,162.82],[0.207608,-0.504777,0.509123,-0.665503],[0,2,-3,0],[9E+09,-27.8948,129.195,9E+09,9E+09,9E+09]];
    PERS robtarget B395S:=[[-109.29,-57.87,162.82],[0.207605,-0.504775,0.509125,-0.665505],[0,2,-3,0],[9E+09,-27.8948,129.195,9E+09,9E+09,9E+09]];

	PERS robtarget G0:=[[0,-168.947,449.567],[0.630104,-0.631581,0.330917,-0.307519],[0,2,-3,0],[9E+09,-1.19001,45.0001,9E+09,9E+09,9E+09]];
	PERS robtarget G1:=[[-93.56,-74.59,-154.76],[0.695032,-0.121449,-0.594906,-0.385055],[-1,0,-2,0],[9E+09,-4.99998,-45,9E+09,9E+09,9E+09]];
	PERS robtarget G2:=[[-94.36,-58.93,-185.09],[0.695028,-0.121442,-0.594905,-0.385066],[-1,0,-2,0],[9E+09,-4.99998,-45,9E+09,9E+09,9E+09]];
	PERS robtarget G3:=[[-93.78,-58.73,-188.84],[0.821373,-0.17617,-0.512082,-0.179116],[-1,0,-2,0],[9E+09,1.02994,-66.6,9E+09,9E+09,9E+09]];
	PERS robtarget G4:=[[-92.88,-36.44,-197.51],[0.815762,-0.177501,-0.507574,-0.21306],[-1,0,-2,0],[9E+09,0.624988,-65.6998,9E+09,9E+09,9E+09]];
	PERS robtarget G5:=[[-90.89,-30.24,-202.73],[0.747426,-0.272864,-0.57506,-0.19028],[-1,0,-2,0],[9E+09,-12.375,-65.6999,9E+09,9E+09,9E+09]];
	PERS robtarget G6:=[[-90.91,-30.79,-207.51],[0.664765,-0.365681,-0.638707,-0.128136],[-1,0,-2,0],[9E+09,-12.375,-65.6998,9E+09,9E+09,9E+09]];
	PERS robtarget G7:=[[-92.77,-31.26,-226.33],[0.738222,-0.273949,-0.571264,-0.2316],[-1,0,-2,0],[9E+09,-15,-57.8636,9E+09,9E+09,9E+09]];
	PERS robtarget G8:=[[-89.55,-20.47,-236.84],[0.806636,-0.157769,-0.506143,-0.26128],[-1,0,-2,0],[9E+09,4.69998,-65.5502,9E+09,9E+09,9E+09]];
	PERS robtarget G9:=[[0,0,0],[0.73728,3.31828E-06,0.675588,2.33895E-06],[0,-1,0,0],[9E+09,9E+09,9E+09,9E+09,9E+09,9E+09]];
	PERS robtarget G10:=[[0,-295.71,565.315],[0.67933,-0.591705,0.324115,-0.288698],[-1,2,-3,0],[9E+09,3.95049,47.5495,9E+09,9E+09,9E+09]];
	PERS robtarget G11:=[[-192.69,-8.97,283.97],[0.00211019,0.781244,-0.624224,3.11178E-05],[0,0,0,0],[9E+09,-20,-20,9E+09,9E+09,9E+09]];
	PERS robtarget G12:=[[191.48,4.49,80.72],[0.00218135,0.703339,-0.710852,2.99839E-05],[0,0,0,0],[9E+09,-7.78641E-06,-4.4762E-05,9E+09,9E+09,9E+09]];
	PERS robtarget G13:=[[-381.15,-11.66,205.25],[0.0462075,0.706542,0.0484395,0.7045],[0,0,-2,0],[9E+09,-7.78641E-06,90,9E+09,9E+09,9E+09]];
	PERS robtarget G14:=[[-326.50,-11.52,205.07],[0.0462054,0.70654,0.0484451,0.704501],[0,0,-2,0],[9E+09,-2.85714E-05,90,9E+09,9E+09,9E+09]];
	PERS robtarget G15:=[[0,-163.407,351.427],[0.678886,-0.563988,0.365725,-0.295427],[0,2,-3,0],[9E+09,5.58454,47.9155,9E+09,9E+09,9E+09]];
	PERS robtarget G16:=[[0,-262.758,400.541],[0.738729,-0.516892,0.334763,-0.273927],[0,2,-3,0],[9E+09,12,49,9E+09,9E+09,9E+09]];
	PERS robtarget G17:=[[0,0,0],[0.73728,3.31828E-06,0.675588,2.33895E-06],[0,-1,0,0],[9E+09,9E+09,9E+09,9E+09,9E+09,9E+09]];
	PERS robtarget G18:=[[0,-145.323,269.777],[0.734056,-0.537733,0.323469,-0.259562],[0,2,-3,0],[9E+09,13.3167,49.1833,9E+09,9E+09,9E+09]];
    PERS robtarget G19:=[[0,-135.956,241.468],[0.72991,-0.487855,0.386257,-0.282905],[0,2,-3,0],[9E+09,14.1988,49.3013,9E+09,9E+09,9E+09]];
    PERS robtarget G195:=[[-109.76,-33.26,246.91],[0.623635,-0.612792,0.3314,-0.354598],[0,2,-3,0],[9E+09,16.8632,49.6371,9E+09,9E+09,9E+09]];
    PERS robtarget G195L:=[[-110.87,-33.62,209.60],[0.626384,-0.615299,0.326701,-0.349739],[0,2,-3,0],[9E+09,16.8632,49.6368,9E+09,9E+09,9E+09]];
    PERS robtarget G195S:=[[-139.94,-19.32,135.81],[0.486218,-0.684613,0.128269,-0.52768],[0,1,-2,0],[9E+09,16.8632,49.6368,9E+09,9E+09,9E+09]];
    PERS robtarget G195R:=[[-141.04,-20.66,117.89],[0.514024,-0.639298,0.122482,-0.558639],[0,1,-2,0],[9E+09,16.8632,49.6368,9E+09,9E+09,9E+09]];
	PERS robtarget G20:=[[192.08,-8.78,283.74],[0.0021613,0.781238,-0.624231,-1.93188E-05],[0,1,-1,0],[9E+09,-20,-20,9E+09,9E+09,9E+09]];
	PERS robtarget G21:=[[0,-171.569,460.423],[0.630145,-0.625031,0.333545,-0.317806],[0,2,-3,0],[9E+09,-0.207117,45.707,9E+09,9E+09,9E+09]];
	PERS robtarget G22:=[[191.48,4.49,80.72],[0.00218135,0.703339,-0.710852,2.99839E-05],[0,0,0,0],[9E+09,-7.78641E-06,-4.4762E-05,9E+09,9E+09,9E+09]];
	PERS robtarget G23:=[[0,-276.741,899.549],[0.552203,-0.714654,0.268259,-0.335229],[-1,1,-2,0],[9E+09,-9.39445,48.6055,9E+09,9E+09,9E+09]];
	PERS robtarget G24:=[[-112.244,-11.52,205.07],[0.0462054,0.70654,0.0484451,0.704501],[0,0,-2,0],[9E+09,-2.85714E-05,90,9E+09,9E+09,9E+09]];
	PERS robtarget G25:=[[0,-154.808,590.675],[0.551243,-0.687236,0.305432,-0.361316],[-1,1,-2,0],[9E+09,-8.9645,48.5355,9E+09,9E+09,9E+09]];
	PERS robtarget G26:=[[-114.082,0,0],[0.73728,3.31828E-06,0.675588,2.33895E-06],[0,-1,0,0],[9E+09,9E+09,9E+09,9E+09,9E+09,9E+09]];
	PERS robtarget G27:=[[0,-225.434,1059.46],[0.495996,-0.745061,0.240573,-0.375496],[-1,1,-2,0],[9E+09,-17.7566,49.7434,9E+09,9E+09,9E+09]];
	PERS robtarget G28:=[[-114.082,0,0],[0.73728,3.31828E-06,0.675588,2.33895E-06],[0,-1,0,0],[9E+09,9E+09,9E+09,9E+09,9E+09,9E+09]];
    PERS robtarget G29:=[[0,-110.494,725.333],[0.468661,-0.74378,0.276228,-0.38839],[-1,1,-2,0],[9E+09,-18.2042,49.7958,9E+09,9E+09,9E+09]];

    PERS robtarget G98:=[[0,0,0],[0.73728,3.31828E-06,0.675588,2.33895E-06],[0,-1,0,0],[9E+09,-24.96,38.42,9E+09,9E+09,9E+09]];
    PERS robtarget G99:=[[0,0,0],[0.73728,3.31828E-06,0.675588,2.33895E-06],[0,-1,0,0],[9E+09,9E+09,9E+09,9E+09,9E+09,9E+09]];

	PERS robtarget H0:=[[0,-166.986,449.528],[0.640484,-0.619834,-0.330146,0.310787],[0,2,-3,0],[9E+09,-1.19003,-45,9E+09,9E+09,9E+09]];
	PERS robtarget H1:=[[90.64,-72.27,-156.11],[0.752512,-0.532327,0.331291,-0.201492],[-1,1,-2,0],[9E+09,-4.99999,44.9999,9E+09,9E+09,9E+09]];
	PERS robtarget H2:=[[88.90,-60.04,-183.51],[0.752508,-0.532326,0.331306,-0.201488],[-1,1,-2,0],[9E+09,-4.99998,45,9E+09,9E+09,9E+09]];
	PERS robtarget H3:=[[90.45,-58.71,-188.66],[0.794107,-0.393028,0.326565,-0.329057],[-1,1,-3,0],[9E+09,1.02999,67.4001,9E+09,9E+09,9E+09]];
	PERS robtarget H4:=[[90.30,-33.99,-198.48],[0.789629,-0.416761,0.307018,-0.329448],[-1,1,-3,0],[9E+09,1.02996,67.4001,9E+09,9E+09,9E+09]];
	PERS robtarget H5:=[[85.59,-30.29,-202.94],[0.725645,-0.533693,0.32099,-0.292535],[-1,1,-3,0],[9E+09,-6.00001,68.3002,9E+09,9E+09,9E+09]];
	PERS robtarget H6:=[[86.14,-29.31,-206.80],[0.630535,-0.629651,0.418595,-0.175339],[-1,1,-2,0],[9E+09,-12.375,68.3,9E+09,9E+09,9E+09]];
	PERS robtarget H7:=[[89.58,-31.11,-224.38],[0.709219,-0.602304,0.289993,-0.223923],[-1,1,-2,0],[9E+09,-15,58.6114,9E+09,9E+09,9E+09]];
	PERS robtarget H8:=[[86.68,-20.53,-235.88],[0.839531,-0.408653,0.28856,-0.211952],[-1,1,-3,0],[9E+09,7.23955,48.7164,9E+09,9E+09,9E+09]];
	PERS robtarget H9:=[[0,0,0],[0.73728,3.31828E-06,0.675588,2.33895E-06],[0,-1,0,0],[9E+09,9E+09,9E+09,9E+09,9E+09,9E+09]];
	PERS robtarget H10:=[[0,-286.11,565.315],[0.684982,-0.582869,-0.326379,0.290757],[-1,1,-2,0],[9E+09,3.95049,-47.5495,9E+09,9E+09,9E+09]];
	PERS robtarget H11:=[[-192.69,-8.97,283.97],[0.00211019,0.781244,-0.624224,3.11178E-05],[0,0,0,0],[9E+09,-20,-20,9E+09,9E+09,9E+09]];
	PERS robtarget H12:=[[191.48,4.49,80.72],[0.00218135,0.703339,-0.710852,2.99839E-05],[0,0,0,0],[9E+09,-7.78641E-06,-4.4762E-05,9E+09,9E+09,9E+09]];
	PERS robtarget H13:=[[-381.15,-11.66,205.25],[0.0462075,0.706542,0.0484395,0.7045],[0,0,-2,0],[9E+09,-7.78641E-06,90,9E+09,9E+09,9E+09]];
	PERS robtarget H14:=[[-326.50,-11.52,205.07],[0.0462054,0.70654,0.0484451,0.704501],[0,0,-2,0],[9E+09,-2.85714E-05,90,9E+09,9E+09,9E+09]];
	PERS robtarget H15:=[[0,-160.551,351.557],[0.685608,-0.56682,-0.355687,0.286606],[0,1,-2,0],[9E+09,5.58452,-47.9155,9E+09,9E+09,9E+09]];
	PERS robtarget H16:=[[0,-253.158,400.541],[0.715385,-0.533731,-0.35774,0.27455],[-1,1,-2,0],[9E+09,12,-49,9E+09,9E+09,9E+09]];
	PERS robtarget H17:=[[0,0,0],[0.73728,3.31828E-06,0.675588,2.33895E-06],[0,-1,0,0],[9E+09,9E+09,9E+09,9E+09,9E+09,9E+09]];
	PERS robtarget H18:=[[0,-135.723,269.777],[0.736141,-0.519694,-0.337867,0.271771],[0,1,-3,0],[9E+09,13.3167,-49.1833,9E+09,9E+09,9E+09]];
    PERS robtarget H19:=[[0,-133.603,241.471],[0.739072,-0.478642,-0.380461,0.282708],[0,1,-2,0],[9E+09,14.1988,-49.3012,9E+09,9E+09,9E+09]];

    PERS robtarget H195:=[[109.27,-30.54,250.10],[0.636823,-0.608095,-0.321054,0.348713],[0,1,-2,0],[9E+09,16.8632,-49.6368,9E+09,9E+09,9E+09]];
    PERS robtarget H195L:=[[110.71,-31.41,207.74],[0.636714,-0.607985,-0.321257,0.348917],[0,1,-2,0],[9E+09,16.8632,-49.6366,9E+09,9E+09,9E+09]];
    PERS robtarget H195S:=[[140.72,-18.83,128.86],[0.660235,-0.505425,-0.44949,0.326489],[0,1,-2,0],[9E+09,16.8632,-49.6368,9E+09,9E+09,9E+09]];
    PERS robtarget H195R:=[[143.21,-20.17,116.33],[0.679562,-0.477178,-0.478781,0.285073],[0,1,-2,0],[9E+09,16.8632,-49.6368,9E+09,9E+09,9E+09]];
	PERS robtarget H20:=[[192.08,-8.78,283.74],[0.0021613,0.781238,-0.624231,-1.93188E-05],[0,1,-1,0],[9E+09,-20,-20,9E+09,9E+09,9E+09]];
	PERS robtarget H21:=[[0,-168.298,460.467],[0.634567,-0.627818,-0.323819,0.313544],[0,2,-3,0],[9E+09,-0.207107,-45.7071,9E+09,9E+09,9E+09]];
	PERS robtarget H22:=[[191.48,4.49,80.72],[0.00218135,0.703339,-0.710852,2.99839E-05],[0,0,0,0],[9E+09,-7.78641E-06,-4.4762E-05,9E+09,9E+09,9E+09]];
	PERS robtarget H23:=[[0,-267.141,899.549],[0.533861,-0.715971,-0.281604,0.350823],[-1,1,-2,0],[9E+09,-9.39445,-48.6055,9E+09,9E+09,9E+09]];
	PERS robtarget H24:=[[108.941,-11.52,205.07],[0.0462054,0.70654,0.0484451,0.704501],[0,0,-2,0],[9E+09,-2.85714E-05,90,9E+09,9E+09,9E+09]];
	PERS robtarget H25:=[[0,-150.669,589.732],[0.559013,-0.684005,-0.301065,0.359168],[-1,2,-3,0],[9E+09,-8.96447,-48.5355,9E+09,9E+09,9E+09]];
	PERS robtarget H26:=[[108.507,0,0],[0.73728,3.31828E-06,0.675588,2.33895E-06],[0,-1,0,0],[9E+09,9E+09,9E+09,9E+09,9E+09,9E+09]];
	PERS robtarget H27:=[[0,-215.834,1059.46],[0.488348,-0.751376,-0.24976,0.366838],[-1,2,-3,0],[9E+09,-17.7566,-49.7434,9E+09,9E+09,9E+09]];
	PERS robtarget H28:=[[108.507,0,0],[0.73728,3.31828E-06,0.675588,2.33895E-06],[0,-1,0,0],[9E+09,9E+09,9E+09,9E+09,9E+09,9E+09]];
    PERS robtarget H29:=[[0,-104.83,722.92],[0.469847,-0.75144,-0.278556,0.37012],[-1,2,-3,0],[9E+09,-18.2042,-49.7957,9E+09,9E+09,9E+09]];

	PERS robtarget G40:=[[-108.94,-15.86,-156.96],[0.675675,-0.591983,0.301839,-0.319237],[-1,1,-2,0],[9E+09,-23.5,50.1962,9E+09,9E+09,9E+09]];
	PERS robtarget G41:=[[-109.84,-16.08,-182.52],[0.632734,-0.641191,0.320266,-0.293176],[-1,1,-2,0],[9E+09,-23.5,50.1962,9E+09,9E+09,9E+09]];
	PERS robtarget G42:=[[-108.39,-15.08,-212.21],[0.62742,-0.644781,0.323279,-0.293414],[-1,1,-2,0],[9E+09,-22,50.1962,9E+09,9E+09,9E+09]];
	PERS robtarget G43:=[[-142.54,1.02,-176.69],[0.536052,-0.432632,0.552635,-0.46912],[-1,1,-2,0],[9E+09,-2.85714E-05,90.0001,9E+09,9E+09,9E+09]];
	PERS robtarget G44:=[[-143.23,-2.89,-180.13],[0.536014,-0.432631,0.552655,-0.469141],[-1,1,-2,0],[9E+09,2.3391E-05,90,9E+09,9E+09,9E+09]];
	PERS robtarget G45:=[[-145.38,-10.22,-212.32],[0.519143,-0.421909,0.568953,-0.478308],[-1,1,-2,0],[9E+09,2.3391E-05,96,9E+09,9E+09,9E+09]];
	PERS robtarget G46:=[[-146.52,-10.10,-258.78],[0.519155,-0.421914,0.568944,-0.478301],[-1,1,-2,0],[9E+09,3.99997,90,9E+09,9E+09,9E+09]];
	PERS robtarget G47:=[[-132.86,0.28,-268.42],[0.590087,-0.522356,0.205632,-0.580223],[-1,1,-3,0],[9E+09,4.99959,90,9E+09,9E+09,9E+09]];
	PERS robtarget G48:=[[-133.49,-1.71,-261.65],[0.580186,-0.451357,0.244207,-0.632475],[-1,1,-3,0],[9E+09,4.99957,89.9999,9E+09,9E+09,9E+09]];
    PERS robtarget G49:=[[-131.64,-7.79,-263.35],[0.598128,-0.383206,0.244438,-0.660037],[-1,1,-3,0],[9E+09,4.99974,90.0001,9E+09,9E+09,9E+09]];

	PERS robtarget G50:=[[-108.25,-80.62,-148.52],[0.585035,-0.4191,0.543218,-0.432441],[-1,1,-2,0],[9E+09,2,81,9E+09,9E+09,9E+09]];
	PERS robtarget G51:=[[-115.24,-74.46,-149.69],[0.396921,-0.583562,0.45899,-0.539664],[-1,-4,2,0],[9E+09,0,90.0003,9E+09,9E+09,9E+09]];
	PERS robtarget G52:=[[-116.08,-29.03,-160.97],[0.396922,-0.583563,0.458992,-0.539661],[-1,-4,2,0],[9E+09,-6.00001,90.0003,9E+09,9E+09,9E+09]];
	PERS robtarget G53:=[[-116.43,-24.84,-162.77],[0.478002,-0.652778,0.396204,-0.43407],[-1,-3,2,0],[9E+09,-6.00003,90.0003,9E+09,9E+09,9E+09]];
	PERS robtarget G54:=[[-106.76,-84.27,-179.76],[0.238217,0.614612,-0.322519,-0.679329],[-1,-1,-3,0],[9E+09,3.60003,-82.9999,9E+09,9E+09,9E+09]];
	PERS robtarget G55:=[[-103.31,-32.44,-190.63],[0.00747561,0.616831,-0.302282,-0.726698],[-1,-1,-3,0],[9E+09,3.00007,-83.0001,9E+09,9E+09,9E+09]];
	PERS robtarget G56:=[[-116.72,-23.97,-161.45],[0.523028,-0.608829,0.331017,-0.496183],[-1,-3,2,0],[9E+09,0.00274881,90.0001,9E+09,9E+09,9E+09]];
	PERS robtarget G57:=[[-116.73,-26.72,-159.83],[0.47391,-0.571518,0.388943,-0.545435],[-1,-3,2,0],[9E+09,0.00274881,90.0002,9E+09,9E+09,9E+09]];
	PERS robtarget G58:=[[-116.06,-74.03,-148.32],[0.473907,-0.571519,0.388945,-0.545436],[-1,-3,2,0],[9E+09,0.00274881,90.0002,9E+09,9E+09,9E+09]];
    PERS robtarget G59:=[[-98.06,-15.53,-192.61],[0.0535957,-0.570788,0.297023,0.763615],[-1,-1,-3,0],[9E+09,-2.00001,-83.0001,9E+09,9E+09,9E+09]];

